  LIN {X 12449.921,Y 0.097,Z 67.094,A 90.00334,B 0.00000,C 180.00000} ; retreat
  ; Step 449, bar 1033
  LIN {X 12465.921,Y 0.097,Z 912.668,A 90.00334,B 0.00000,C 180.00000} ; outside
  LIN {X 12465.921,Y 0.097,Z 17.094,A 90.00334,B 0.00000,C 180.00000} ; preinsert
  LIN {X 12465.921,Y 0.097,Z -232.906,A 90.00334,B 0.00000,C 180.00000} ; insert
  LIN {X 12465.921,Y 0.097,Z -232.906,A 90.00334,B 0.00000,C 180.00000} ; release
  LIN {X 12465.921,Y 0.097,Z 67.094,A 90.00334,B 0.00000,C 180.00000} ; retreat
  ; Step 450, bar 295
  LIN {X 0.000,Y -2325.000,Z 1045.621,A 0.00000,B 0.00000,C 180.00000} ; outside
  LIN {X 0.000,Y -2325.000,Z 147.121,A 0.00000,B 0.00000,C 180.00000} ; preinsert
  LIN {X 0.000,Y -2325.000,Z -102.879,A 0.00000,B 0.00000,C 180.00000} ; insert
  LIN {X 0.000,Y -2325.000,Z -102.879,A 0.00000,B 0.00000,C 180.00000} ; release
  LIN {X 0.000,Y -2325.000,Z 197.121,A 0.00000,B 0.00000,C 180.00000} ; retreat
  ; Step 451, bar 322
  LIN {X 0.000,Y 2325.000,Z 1045.621,A 0.00000,B 0.00000,C 180.00000} ; outside
  LIN {X 0.000,Y 2325.000,Z 147.121,A 0.00000,B 0.00000,C 180.00000} ; preinsert
  LIN {X 0.000,Y 2325.000,Z -102.879,A 0.00000,B 0.00000,C 180.00000} ; insert
  LIN {X 0.000,Y 2325.000,Z -102.879,A 0.00000,B 0.00000,C 180.00000} ; release
  LIN {X 0.000,Y 2325.000,Z 197.121,A 0.00000,B 0.00000,C 180.00000} ; retreat
  ; Step 452, bar 293
  LIN {X 0.000,Y -1977.000,Z 1051.871,A 0.00000,B 0.00000,C 180.00000} ; outside
  LIN {X 0.000,Y -1977.000,Z 150.246,A 0.00000,B 0.00000,C 180.00000} ; preinsert
  LIN {X 0.000,Y -1977.000,Z -99.754,A 0.00000,B 0.00000,C 180.00000} ; insert
  LIN {X 0.000,Y -1977.000,Z -99.754,A 0.00000,B 0.00000,C 180.00000} ; release
  LIN {X 0.000,Y -1977.000,Z 200.246,A 0.00000,B 0.00000,C 180.00000} ; retreat
  ; Step 453, bar 320
  LIN {X 0.000,Y 1977.000,Z 1051.871,A 0.00000,B 0.00000,C 180.00000} ; outside
  LIN {X 0.000,Y 1977.000,Z 150.246,A 0.00000,B 0.00000,C 180.00000} ; preinsert
  LIN {X 0.000,Y 1977.000,Z -99.754,A 0.00000,B 0.00000,C 180.00000} ; insert
  LIN {X 0.000,Y 1977.000,Z -99.754,A 0.00000,B 0.00000,C 180.00000} ; release
  LIN {X 0.000,Y 1977.000,Z 200.246,A 0.00000,B 0.00000,C 180.00000} ; retreat
  ; Step 454, bar 294
  LIN {X 0.484,Y -2151.056,Z 1053.018,A -179.99813,B 0.00000,C 180.00000} ; outside
  LIN {X 0.484,Y -2151.056,Z 150.800,A -179.99813,B 0.00000,C 180.00000} ; preinsert
  LIN {X 0.484,Y -2151.056,Z -99.200,A -179.99813,B 0.00000,C 180.00000} ; insert
  LIN {X 0.484,Y -2151.056,Z -99.200,A -179.99813,B 0.00000,C 180.00000} ; release
  LIN {X 0.484,Y -2151.056,Z 200.800,A -179.99813,B 0.00000,C 180.00000} ; retreat
  ; Step 455, bar 1893
  LIN {X 3995.484,Y -2151.056,Z 1053.018,A -179.99813,B 0.00000,C 180.00000} ; outside
  LIN {X 3995.484,Y -2151.056,Z 150.800,A -179.99813,B 0.00000,C 180.00000} ; preinsert
  LIN {X 3995.484,Y -2151.056,Z -99.200,A -179.99813,B 0.00000,C 180.00000} ; insert
  LIN {X 3995.484,Y -2151.056,Z -99.200,A -179.99813,B 0.00000,C 180.00000} ; release
  LIN {X 3995.484,Y -2151.056,Z 200.800,A -179.99813,B 0.00000,C 180.00000} ; retreat
  ; Step 456, bar 1897
  LIN {X 7995.484,Y -2151.056,Z 1053.018,A -179.99813,B 0.00000,C 180.00000} ; outside
  LIN {X 7995.484,Y -2151.056,Z 150.800,A -179.99813,B 0.00000,C 180.00000} ; preinsert
  LIN {X 7995.484,Y -2151.056,Z -99.200,A -179.99813,B 0.00000,C 180.00000} ; insert
  LIN {X 7995.484,Y -2151.056,Z -99.200,A -179.99813,B 0.00000,C 180.00000} ; release
  LIN {X 7995.484,Y -2151.056,Z 200.800,A -179.99813,B 0.00000,C 180.00000} ; retreat
  ; Step 457, bar 1905
  LIN {X 11995.484,Y -2151.056,Z 1053.018,A -179.99813,B 0.00000,C 180.00000} ; outside
  LIN {X 11995.484,Y -2151.056,Z 150.800,A -179.99813,B 0.00000,C 180.00000} ; preinsert
  LIN {X 11995.484,Y -2151.056,Z -99.200,A -179.99813,B 0.00000,C 180.00000} ; insert
  LIN {X 11995.484,Y -2151.056,Z -99.200,A -179.99813,B 0.00000,C 180.00000} ; release
  LIN {X 11995.484,Y -2151.056,Z 200.800,A -179.99813,B 0.00000,C 180.00000} ; retreat
  ; Step 458, bar 1922
  LIN {X -11995.484,Y 2151.056,Z 1053.018,A 0.00187,B 0.00000,C 180.00000} ; outside
  LIN {X -11995.484,Y 2151.056,Z 150.800,A 0.00187,B 0.00000,C 180.00000} ; preinsert
  LIN {X -11995.484,Y 2151.056,Z -99.200,A 0.00187,B 0.00000,C 180.00000} ; insert
  LIN {X -11995.484,Y 2151.056,Z -99.200,A 0.00187,B 0.00000,C 180.00000} ; release
  LIN {X -11995.484,Y 2151.056,Z 200.800,A 0.00187,B 0.00000,C 180.00000} ; retreat
  ; Step 459, bar 1914
  LIN {X -7995.484,Y 2151.056,Z 1053.018,A 0.00187,B 0.00000,C 180.00000} ; outside
  LIN {X -7995.484,Y 2151.056,Z 150.800,A 0.00187,B 0.00000,C 180.00000} ; preinsert
  LIN {X -7995.484,Y 2151.056,Z -99.200,A 0.00187,B 0.00000,C 180.00000} ; insert
  LIN {X -7995.484,Y 2151.056,Z -99.200,A 0.00187,B 0.00000,C 180.00000} ; release
  LIN {X -7995.484,Y 2151.056,Z 200.800,A 0.00187,B 0.00000,C 180.00000} ; retreat
  ; Step 460, bar 1910
  LIN {X -3995.484,Y 2151.056,Z 1053.018,A 0.00187,B 0.00000,C 180.00000} ; outside
  LIN {X -3995.484,Y 2151.056,Z 150.800,A 0.00187,B 0.00000,C 180.00000} ; preinsert
  LIN {X -3995.484,Y 2151.056,Z -99.200,A 0.00187,B 0.00000,C 180.00000} ; insert
  LIN {X -3995.484,Y 2151.056,Z -99.200,A 0.00187,B 0.00000,C 180.00000} ; release
  LIN {X -3995.484,Y 2151.056,Z 200.800,A 0.00187,B 0.00000,C 180.00000} ; retreat
  ; Step 461, bar 1921
  LIN {X -11995.484,Y -2151.056,Z 1053.018,A -0.00187,B 0.00000,C 180.00000} ; outside
  LIN {X -11995.484,Y -2151.056,Z 150.800,A -0.00187,B 0.00000,C 180.00000} ; preinsert
  LIN {X -11995.484,Y -2151.056,Z -99.200,A -0.00187,B 0.00000,C 180.00000} ; insert
  LIN {X -11995.484,Y -2151.056,Z -99.200,A -0.00187,B 0.00000,C 180.00000} ; release
  LIN {X -11995.484,Y -2151.056,Z 200.800,A -0.00187,B 0.00000,C 180.00000} ; retreat
  ; Step 462, bar 1913
  LIN {X -7995.484,Y -2151.056,Z 1053.018,A -0.00187,B 0.00000,C 180.00000} ; outside
  LIN {X -7995.484,Y -2151.056,Z 150.800,A -0.00187,B 0.00000,C 180.00000} ; preinsert
  LIN {X -7995.484,Y -2151.056,Z -99.200,A -0.00187,B 0.00000,C 180.00000} ; insert
  LIN {X -7995.484,Y -2151.056,Z -99.200,A -0.00187,B 0.00000,C 180.00000} ; release
  LIN {X -7995.484,Y -2151.056,Z 200.800,A -0.00187,B 0.00000,C 180.00000} ; retreat
  ; Step 463, bar 1909
  LIN {X -3995.484,Y -2151.056,Z 1053.018,A -0.00187,B 0.00000,C 180.00000} ; outside
  LIN {X -3995.484,Y -2151.056,Z 150.800,A -0.00187,B 0.00000,C 180.00000} ; preinsert
  LIN {X -3995.484,Y -2151.056,Z -99.200,A -0.00187,B 0.00000,C 180.00000} ; insert
  LIN {X -3995.484,Y -2151.056,Z -99.200,A -0.00187,B 0.00000,C 180.00000} ; release
  LIN {X -3995.484,Y -2151.056,Z 200.800,A -0.00187,B 0.00000,C 180.00000} ; retreat
  ; Step 464, bar 321
  LIN {X 0.484,Y 2151.056,Z 1053.018,A 179.99813,B 0.00000,C 180.00000} ; outside
  LIN {X 0.484,Y 2151.056,Z 150.800,A 179.99813,B 0.00000,C 180.00000} ; preinsert
  LIN {X 0.484,Y 2151.056,Z -99.200,A 179.99813,B 0.00000,C 180.00000} ; insert
  LIN {X 0.484,Y 2151.056,Z -99.200,A 179.99813,B 0.00000,C 180.00000} ; release
  LIN {X 0.484,Y 2151.056,Z 200.800,A 179.99813,B 0.00000,C 180.00000} ; retreat
  ; Step 465, bar 1894
  LIN {X 3995.484,Y 2151.056,Z 1053.018,A 179.99813,B 0.00000,C 180.00000} ; outside
  LIN {X 3995.484,Y 2151.056,Z 150.800,A 179.99813,B 0.00000,C 180.00000} ; preinsert
  LIN {X 3995.484,Y 2151.056,Z -99.200,A 179.99813,B 0.00000,C 180.00000} ; insert
  LIN {X 3995.484,Y 2151.056,Z -99.200,A 179.99813,B 0.00000,C 180.00000} ; release
  LIN {X 3995.484,Y 2151.056,Z 200.800,A 179.99813,B 0.00000,C 180.00000} ; retreat
  ; Step 466, bar 1898
  LIN {X 7995.484,Y 2151.056,Z 1053.018,A 179.99813,B 0.00000,C 180.00000} ; outside
  LIN {X 7995.484,Y 2151.056,Z 150.800,A 179.99813,B 0.00000,C 180.00000} ; preinsert
  LIN {X 7995.484,Y 2151.056,Z -99.200,A 179.99813,B 0.00000,C 180.00000} ; insert
  LIN {X 7995.484,Y 2151.056,Z -99.200,A 179.99813,B 0.00000,C 180.00000} ; release
  LIN {X 7995.484,Y 2151.056,Z 200.800,A 179.99813,B 0.00000,C 180.00000} ; retreat
  ; Step 467, bar 1906
  LIN {X 11995.484,Y 2151.056,Z 1053.018,A 179.99813,B 0.00000,C 180.00000} ; outside
  LIN {X 11995.484,Y 2151.056,Z 150.800,A 179.99813,B 0.00000,C 180.00000} ; preinsert
  LIN {X 11995.484,Y 2151.056,Z -99.200,A 179.99813,B 0.00000,C 180.00000} ; insert
  LIN {X 11995.484,Y 2151.056,Z -99.200,A 179.99813,B 0.00000,C 180.00000} ; release
  LIN {X 11995.484,Y 2151.056,Z 200.800,A 179.99813,B 0.00000,C 180.00000} ; retreat
  ; Step 468, bar 1923
  LIN {X -11994.516,Y -2150.911,Z 797.364,A -179.99813,B 0.00000,C -180.00000} ; outside
  LIN {X -11994.516,Y -2150.911,Z -105.285,A -179.99813,B 0.00000,C -180.00000} ; preinsert
  LIN {X -11994.516,Y -2150.911,Z -355.285,A -179.99813,B 0.00000,C -180.00000} ; insert
  LIN {X -11994.516,Y -2150.911,Z -355.285,A -179.99813,B 0.00000,C -180.00000} ; release
  LIN {X -11994.516,Y -2150.911,Z -55.285,A -179.99813,B 0.00000,C -180.00000} ; retreat
  ; Step 469, bar 1915
  LIN {X -7994.516,Y -2150.911,Z 797.364,A -179.99813,B 0.00000,C -180.00000} ; outside
  LIN {X -7994.516,Y -2150.911,Z -105.285,A -179.99813,B 0.00000,C -180.00000} ; preinsert
  LIN {X -7994.516,Y -2150.911,Z -355.285,A -179.99813,B 0.00000,C -180.00000} ; insert
  LIN {X -7994.516,Y -2150.911,Z -355.285,A -179.99813,B 0.00000,C -180.00000} ; release
  LIN {X -7994.516,Y -2150.911,Z -55.285,A -179.99813,B 0.00000,C -180.00000} ; retreat
  ; Step 470, bar 1899
  LIN {X 7994.516,Y -2150.911,Z 797.364,A -0.00187,B 0.00000,C 180.00000} ; outside
  LIN {X 7994.516,Y -2150.911,Z -105.285,A -0.00187,B 0.00000,C 180.00000} ; preinsert
  LIN {X 7994.516,Y -2150.911,Z -355.285,A -0.00187,B 0.00000,C 180.00000} ; insert
  LIN {X 7994.516,Y -2150.911,Z -355.285,A -0.00187,B 0.00000,C 180.00000} ; release
  LIN {X 7994.516,Y -2150.911,Z -55.285,A -0.00187,B 0.00000,C 180.00000} ; retreat
  ; Step 471, bar 1907
  LIN {X 11994.516,Y -2150.911,Z 797.364,A -0.00187,B 0.00000,C 180.00000} ; outside
  LIN {X 11994.516,Y -2150.911,Z -105.285,A -0.00187,B 0.00000,C 180.00000} ; preinsert
  LIN {X 11994.516,Y -2150.911,Z -355.285,A -0.00187,B 0.00000,C 180.00000} ; insert
  LIN {X 11994.516,Y -2150.911,Z -355.285,A -0.00187,B 0.00000,C 180.00000} ; release
  LIN {X 11994.516,Y -2150.911,Z -55.285,A -0.00187,B 0.00000,C 180.00000} ; retreat
  ; Step 472, bar 1911
  LIN {X -3994.516,Y -2150.911,Z 797.364,A -179.99813,B 0.00000,C -180.00000} ; outside
  LIN {X -3994.516,Y -2150.911,Z -105.285,A -179.99813,B 0.00000,C -180.00000} ; preinsert
  LIN {X -3994.516,Y -2150.911,Z -355.285,A -179.99813,B 0.00000,C -180.00000} ; insert
  LIN {X -3994.516,Y -2150.911,Z -355.285,A -179.99813,B 0.00000,C -180.00000} ; release
  LIN {X -3994.516,Y -2150.911,Z -55.285,A -179.99813,B 0.00000,C -180.00000} ; retreat
  ; Step 473, bar 1861
  LIN {X -0.484,Y -2150.911,Z 797.364,A -0.00187,B 0.00000,C 180.00000} ; outside
  LIN {X -0.484,Y -2150.911,Z -105.285,A -0.00187,B 0.00000,C 180.00000} ; preinsert
  LIN {X -0.484,Y -2150.911,Z -355.285,A -0.00187,B 0.00000,C 180.00000} ; insert
  LIN {X -0.484,Y -2150.911,Z -355.285,A -0.00187,B 0.00000,C 180.00000} ; release
  LIN {X -0.484,Y -2150.911,Z -55.285,A -0.00187,B 0.00000,C 180.00000} ; retreat
  ; Step 474, bar 1895
  LIN {X 3994.516,Y -2150.911,Z 797.364,A -0.00187,B 0.00000,C 180.00000} ; outside
  LIN {X 3994.516,Y -2150.911,Z -105.285,A -0.00187,B 0.00000,C 180.00000} ; preinsert
  LIN {X 3994.516,Y -2150.911,Z -355.285,A -0.00187,B 0.00000,C 180.00000} ; insert
  LIN {X 3994.516,Y -2150.911,Z -355.285,A -0.00187,B 0.00000,C 180.00000} ; release
  LIN {X 3994.516,Y -2150.911,Z -55.285,A -0.00187,B 0.00000,C 180.00000} ; retreat
  ; Step 475, bar 1924
  LIN {X -11994.516,Y 2150.911,Z 797.364,A 179.99813,B 0.00000,C -180.00000} ; outside
  LIN {X -11994.516,Y 2150.911,Z -105.285,A 179.99813,B 0.00000,C -180.00000} ; preinsert
  LIN {X -11994.516,Y 2150.911,Z -355.285,A 179.99813,B 0.00000,C -180.00000} ; insert
  LIN {X -11994.516,Y 2150.911,Z -355.285,A 179.99813,B 0.00000,C -180.00000} ; release
  LIN {X -11994.516,Y 2150.911,Z -55.285,A 179.99813,B 0.00000,C -180.00000} ; retreat
  ; Step 476, bar 1916
  LIN {X -7994.516,Y 2150.911,Z 797.364,A 179.99813,B 0.00000,C -180.00000} ; outside
  LIN {X -7994.516,Y 2150.911,Z -105.285,A 179.99813,B 0.00000,C -180.00000} ; preinsert
  LIN {X -7994.516,Y 2150.911,Z -355.285,A 179.99813,B 0.00000,C -180.00000} ; insert
  LIN {X -7994.516,Y 2150.911,Z -355.285,A 179.99813,B 0.00000,C -180.00000} ; release
  LIN {X -7994.516,Y 2150.911,Z -55.285,A 179.99813,B 0.00000,C -180.00000} ; retreat
  ; Step 477, bar 1900
  LIN {X 7994.516,Y 2150.911,Z 797.364,A 0.00187,B 0.00000,C 180.00000} ; outside
  LIN {X 7994.516,Y 2150.911,Z -105.285,A 0.00187,B 0.00000,C 180.00000} ; preinsert
  LIN {X 7994.516,Y 2150.911,Z -355.285,A 0.00187,B 0.00000,C 180.00000} ; insert
  LIN {X 7994.516,Y 2150.911,Z -355.285,A 0.00187,B 0.00000,C 180.00000} ; release
  LIN {X 7994.516,Y 2150.911,Z -55.285,A 0.00187,B 0.00000,C 180.00000} ; retreat
  ; Step 478, bar 1908
  LIN {X 11994.516,Y 2150.911,Z 797.364,A 0.00187,B 0.00000,C 180.00000} ; outside
  LIN {X 11994.516,Y 2150.911,Z -105.285,A 0.00187,B 0.00000,C 180.00000} ; preinsert
  LIN {X 11994.516,Y 2150.911,Z -355.285,A 0.00187,B 0.00000,C 180.00000} ; insert
  LIN {X 11994.516,Y 2150.911,Z -355.285,A 0.00187,B 0.00000,C 180.00000} ; release
  LIN {X 11994.516,Y 2150.911,Z -55.285,A 0.00187,B 0.00000,C 180.00000} ; retreat
  ; Step 479, bar 1912
  LIN {X -3994.516,Y 2150.911,Z 797.364,A 179.99813,B 0.00000,C -180.00000} ; outside
  LIN {X -3994.516,Y 2150.911,Z -105.285,A 179.99813,B 0.00000,C -180.00000} ; preinsert
  LIN {X -3994.516,Y 2150.911,Z -355.285,A 179.99813,B 0.00000,C -180.00000} ; insert
  LIN {X -3994.516,Y 2150.911,Z -355.285,A 179.99813,B 0.00000,C -180.00000} ; release
  LIN {X -3994.516,Y 2150.911,Z -55.285,A 179.99813,B 0.00000,C -180.00000} ; retreat
  ; Step 480, bar 1874
  LIN {X -0.484,Y 2150.911,Z 797.364,A 0.00187,B 0.00000,C 180.00000} ; outside
  LIN {X -0.484,Y 2150.911,Z -105.285,A 0.00187,B 0.00000,C 180.00000} ; preinsert
  LIN {X -0.484,Y 2150.911,Z -355.285,A 0.00187,B 0.00000,C 180.00000} ; insert
  LIN {X -0.484,Y 2150.911,Z -355.285,A 0.00187,B 0.00000,C 180.00000} ; release
  LIN {X -0.484,Y 2150.911,Z -55.285,A 0.00187,B 0.00000,C 180.00000} ; retreat
  ; Step 481, bar 1896
  LIN {X 3994.516,Y 2150.911,Z 797.364,A 0.00187,B 0.00000,C 180.00000} ; outside
  LIN {X 3994.516,Y 2150.911,Z -105.285,A 0.00187,B 0.00000,C 180.00000} ; preinsert
  LIN {X 3994.516,Y 2150.911,Z -355.285,A 0.00187,B 0.00000,C 180.00000} ; insert
  LIN {X 3994.516,Y 2150.911,Z -355.285,A 0.00187,B 0.00000,C 180.00000} ; release
  LIN {X 3994.516,Y 2150.911,Z -55.285,A 0.00187,B 0.00000,C 180.00000} ; retreat
  ; Step 482, bar 1917
  LIN {X -15308.088,Y -2150.945,Z 1052.784,A -0.00257,B 0.00000,C 180.00000} ; outside
  LIN {X -15308.088,Y -2150.945,Z 150.678,A -0.00257,B 0.00000,C 180.00000} ; preinsert
  LIN {X -15308.088,Y -2150.945,Z -99.322,A -0.00257,B 0.00000,C 180.00000} ; insert
  LIN {X -15308.088,Y -2150.945,Z -99.322,A -0.00257,B 0.00000,C 180.00000} ; release
  LIN {X -15308.088,Y -2150.945,Z 200.678,A -0.00257,B 0.00000,C 180.00000} ; retreat
  ; Step 483, bar 1901
  LIN {X 15308.088,Y -2150.945,Z 1052.784,A -179.99743,B 0.00000,C 180.00000} ; outside
  LIN {X 15308.088,Y -2150.945,Z 150.678,A -179.99743,B 0.00000,C 180.00000} ; preinsert
  LIN {X 15308.088,Y -2150.945,Z -99.322,A -179.99743,B 0.00000,C 180.00000} ; insert
  LIN {X 15308.088,Y -2150.945,Z -99.322,A -179.99743,B 0.00000,C 180.00000} ; release
  LIN {X 15308.088,Y -2150.945,Z 200.678,A -179.99743,B 0.00000,C 180.00000} ; retreat
  ; Step 484, bar 1918
  LIN {X -15308.088,Y 2150.945,Z 1052.784,A 0.00257,B 0.00000,C 180.00000} ; outside
  LIN {X -15308.088,Y 2150.945,Z 150.678,A 0.00257,B 0.00000,C 180.00000} ; preinsert
  LIN {X -15308.088,Y 2150.945,Z -99.322,A 0.00257,B 0.00000,C 180.00000} ; insert
  LIN {X -15308.088,Y 2150.945,Z -99.322,A 0.00257,B 0.00000,C 180.00000} ; release
  LIN {X -15308.088,Y 2150.945,Z 200.678,A 0.00257,B 0.00000,C 180.00000} ; retreat
  ; Step 485, bar 1902
  LIN {X 15308.088,Y 2150.945,Z 1052.784,A 179.99743,B 0.00000,C -180.00000} ; outside
  LIN {X 15308.088,Y 2150.945,Z 150.678,A 179.99743,B 0.00000,C -180.00000} ; preinsert
  LIN {X 15308.088,Y 2150.945,Z -99.322,A 179.99743,B 0.00000,C -180.00000} ; insert
  LIN {X 15308.088,Y 2150.945,Z -99.322,A 179.99743,B 0.00000,C -180.00000} ; release
  LIN {X 15308.088,Y 2150.945,Z 200.678,A 179.99743,B 0.00000,C -180.00000} ; retreat
  ; Step 486, bar 1852
  LIN {X -16250.000,Y -0.156,Z 909.110,A 90.00000,B 0.00000,C 180.00000} ; outside
  LIN {X -16250.000,Y -0.156,Z 7.730,A 90.00000,B 0.00000,C 180.00000} ; preinsert
  LIN {X -16250.000,Y -0.156,Z -242.270,A 90.00000,B 0.00000,C 180.00000} ; insert
  LIN {X -16250.000,Y -0.156,Z -242.270,A 90.00000,B 0.00000,C 180.00000} ; release
  LIN {X -16250.000,Y -0.156,Z 57.730,A 90.00000,B 0.00000,C 180.00000} ; retreat
  ; Step 487, bar 1851
  LIN {X -16150.000,Y -0.156,Z 909.110,A 90.00000,B 0.00000,C 180.00000} ; outside
  LIN {X -16150.000,Y -0.156,Z 7.730,A 90.00000,B 0.00000,C 180.00000} ; preinsert
  LIN {X -16150.000,Y -0.156,Z -242.270,A 90.00000,B 0.00000,C 180.00000} ; insert
  LIN {X -16150.000,Y -0.156,Z -242.270,A 90.00000,B 0.00000,C 180.00000} ; release
  LIN {X -16150.000,Y -0.156,Z 57.730,A 90.00000,B 0.00000,C 180.00000} ; retreat
  ; Step 488, bar 1064
  LIN {X 16150.000,Y -0.171,Z 909.110,A 90.00000,B 0.00000,C 180.00000} ; outside
  LIN {X 16150.000,Y -0.171,Z 7.730,A 90.00000,B 0.00000,C 180.00000} ; preinsert
  LIN {X 16150.000,Y -0.171,Z -242.270,A 90.00000,B 0.00000,C 180.00000} ; insert
  LIN {X 16150.000,Y -0.171,Z -242.270,A 90.00000,B 0.00000,C 180.00000} ; release
  LIN {X 16150.000,Y -0.171,Z 57.730,A 90.00000,B 0.00000,C 180.00000} ; retreat
  ; Step 489, bar 1065
  LIN {X 16250.000,Y -0.171,Z 909.110,A 90.00000,B 0.00000,C 180.00000} ; outside
  LIN {X 16250.000,Y -0.171,Z 7.730,A 90.00000,B 0.00000,C 180.00000} ; preinsert
  LIN {X 16250.000,Y -0.171,Z -242.270,A 90.00000,B 0.00000,C 180.00000} ; insert
  LIN {X 16250.000,Y -0.171,Z -242.270,A 90.00000,B 0.00000,C 180.00000} ; release
  LIN {X 16250.000,Y -0.171,Z 57.730,A 90.00000,B 0.00000,C 180.00000} ; retreat
  ; Step 490, bar 1233
  LIN {X -12349.921,Y 0.110,Z 926.030,A 89.99666,B 0.00000,C 180.00000} ; outside
  LIN {X -12349.921,Y 0.110,Z 23.775,A 89.99666,B 0.00000,C 180.00000} ; preinsert
  LIN {X -12349.921,Y 0.110,Z -226.225,A 89.99666,B 0.00000,C 180.00000} ; insert
  LIN {X -12349.921,Y 0.110,Z -226.225,A 89.99666,B 0.00000,C 180.00000} ; release
  LIN {X -12349.921,Y 0.110,Z 73.775,A 89.99666,B 0.00000,C 180.00000} ; retreat
  ; Step 491, bar 1018
  LIN {X 12349.921,Y 0.097,Z 926.030,A 90.00334,B 0.00000,C 180.00000} ; outside
  LIN {X 12349.921,Y 0.097,Z 23.775,A 90.00334,B 0.00000,C 180.00000} ; preinsert
  LIN {X 12349.921,Y 0.097,Z -226.225,A 90.00334,B 0.00000,C 180.00000} ; insert
  LIN {X 12349.921,Y 0.097,Z -226.225,A 90.00334,B 0.00000,C 180.00000} ; release
  LIN {X 12349.921,Y 0.097,Z 73.775,A 90.00334,B 0.00000,C 180.00000} ; retreat
  ; Step 492, bar 2977
  LIN {X -14850.007,Y -1181.237,Z 942.517,A -92.05282,B 0.00000,C -180.00000} ; outside
  LIN {X -14850.007,Y -1181.237,Z 3.500,A -92.05282,B 0.00000,C -180.00000} ; preinsert
  LIN {X -14850.007,Y -1181.237,Z -246.500,A -92.05282,B 0.00000,C -180.00000} ; insert
  LIN {X -14850.007,Y -1181.237,Z -246.500,A -92.05282,B 0.00000,C -180.00000} ; release
  LIN {X -14850.007,Y -1181.237,Z 53.500,A -92.05282,B 0.00000,C -180.00000} ; retreat
  ; Step 493, bar 3016
  LIN {X 14850.007,Y -1181.237,Z 942.518,A -87.94718,B 0.00000,C 180.00000} ; outside
  LIN {X 14850.007,Y -1181.237,Z 3.500,A -87.94718,B 0.00000,C 180.00000} ; preinsert
  LIN {X 14850.007,Y -1181.237,Z -246.500,A -87.94718,B 0.00000,C 180.00000} ; insert
  LIN {X 14850.007,Y -1181.237,Z -246.500,A -87.94718,B 0.00000,C 180.00000} ; release
  LIN {X 14850.007,Y -1181.237,Z 53.500,A -87.94718,B 0.00000,C 180.00000} ; retreat
  ; Step 494, bar 2959
  LIN {X -14850.007,Y 1181.237,Z 942.518,A 92.05282,B 0.00000,C 180.00000} ; outside
  LIN {X -14850.007,Y 1181.237,Z 3.500,A 92.05282,B 0.00000,C 180.00000} ; preinsert
  LIN {X -14850.007,Y 1181.237,Z -246.500,A 92.05282,B 0.00000,C 180.00000} ; insert
  LIN {X -14850.007,Y 1181.237,Z -246.500,A 92.05282,B 0.00000,C 180.00000} ; release
  LIN {X -14850.007,Y 1181.237,Z 53.500,A 92.05282,B 0.00000,C 180.00000} ; retreat
  ; Step 495, bar 2998
  LIN {X 14850.007,Y 1181.237,Z 942.517,A 87.94718,B 0.00000,C 180.00000} ; outside
  LIN {X 14850.007,Y 1181.237,Z 3.500,A 87.94718,B 0.00000,C 180.00000} ; preinsert
  LIN {X 14850.007,Y 1181.237,Z -246.500,A 87.94718,B 0.00000,C 180.00000} ; insert
  LIN {X 14850.007,Y 1181.237,Z -246.500,A 87.94718,B 0.00000,C 180.00000} ; release
  LIN {X 14850.007,Y 1181.237,Z 53.500,A 87.94718,B 0.00000,C 180.00000} ; retreat
  ; Step 496, bar 3011
  LIN {X 14050.059,Y -1181.145,Z 931.267,A 88.24449,B 0.00000,C 180.00000} ; outside
  LIN {X 14050.059,Y -1181.145,Z 14.532,A 88.24449,B 0.00000,C 180.00000} ; preinsert
  LIN {X 14050.059,Y -1181.145,Z -235.468,A 88.24449,B 0.00000,C 180.00000} ; insert
  LIN {X 14050.059,Y -1181.145,Z -235.468,A 88.24449,B 0.00000,C 180.00000} ; release
  LIN {X 14050.059,Y -1181.145,Z 64.532,A 88.24449,B 0.00000,C 180.00000} ; retreat
  ; Step 497, bar 2953
  LIN {X -14050.059,Y 1181.145,Z 931.267,A -91.75551,B 0.00000,C -180.00000} ; outside
  LIN {X -14050.059,Y 1181.145,Z 14.532,A -91.75551,B 0.00000,C -180.00000} ; preinsert
  LIN {X -14050.059,Y 1181.145,Z -235.468,A -91.75551,B 0.00000,C -180.00000} ; insert
  LIN {X -14050.059,Y 1181.145,Z -235.468,A -91.75551,B 0.00000,C -180.00000} ; release
  LIN {X -14050.059,Y 1181.145,Z 64.532,A -91.75551,B 0.00000,C -180.00000} ; retreat
  ; Step 498, bar 2972
  LIN {X -14050.059,Y -1181.145,Z 931.267,A 91.75551,B 0.00000,C 180.00000} ; outside
  LIN {X -14050.059,Y -1181.145,Z 14.532,A 91.75551,B 0.00000,C 180.00000} ; preinsert
  LIN {X -14050.059,Y -1181.145,Z -235.468,A 91.75551,B 0.00000,C 180.00000} ; insert
  LIN {X -14050.059,Y -1181.145,Z -235.468,A 91.75551,B 0.00000,C 180.00000} ; release
  LIN {X -14050.059,Y -1181.145,Z 64.532,A 91.75551,B 0.00000,C 180.00000} ; retreat
  ; Step 499, bar 2992
  LIN {X 14050.059,Y 1181.145,Z 931.267,A -88.24449,B 0.00000,C 180.00000} ; outside
  LIN {X 14050.059,Y 1181.145,Z 14.532,A -88.24449,B 0.00000,C 180.00000} ; preinsert
  LIN {X 14050.059,Y 1181.145,Z -235.468,A -88.24449,B 0.00000,C 180.00000} ; insert
  LIN {X 14050.059,Y 1181.145,Z -235.468,A -88.24449,B 0.00000,C 180.00000} ; release
  LIN {X 14050.059,Y 1181.145,Z 64.532,A -88.24449,B 0.00000,C 180.00000} ; retreat
  ; Step 500, bar 2967
  LIN {X -13249.916,Y -1181.296,Z 955.534,A 87.44234,B 0.00000,C -180.00000} ; outside
  LIN {X -13249.916,Y -1181.296,Z 50.876,A 87.44234,B 0.00000,C -180.00000} ; preinsert
  LIN {X -13249.916,Y -1181.296,Z -199.124,A 87.44234,B 0.00000,C -180.00000} ; insert
  LIN {X -13249.916,Y -1181.296,Z -199.124,A 87.44234,B 0.00000,C -180.00000} ; release
  LIN {X -13249.916,Y -1181.296,Z 100.876,A 87.44234,B 0.00000,C -180.00000} ; retreat
  ; Step 501, bar 2986
  LIN {X 13249.916,Y 1181.296,Z 955.534,A -92.55766,B 0.00000,C -180.00000} ; outside
  LIN {X 13249.916,Y 1181.296,Z 50.876,A -92.55766,B 0.00000,C -180.00000} ; preinsert
  LIN {X 13249.916,Y 1181.296,Z -199.124,A -92.55766,B 0.00000,C -180.00000} ; insert
  LIN {X 13249.916,Y 1181.296,Z -199.124,A -92.55766,B 0.00000,C -180.00000} ; release
  LIN {X 13249.916,Y 1181.296,Z 100.876,A -92.55766,B 0.00000,C -180.00000} ; retreat
  ; Step 502, bar 3006
  LIN {X 13249.916,Y -1181.296,Z 955.534,A 92.55766,B 0.00000,C 180.00000} ; outside
  LIN {X 13249.916,Y -1181.296,Z 50.876,A 92.55766,B 0.00000,C 180.00000} ; preinsert
  LIN {X 13249.916,Y -1181.296,Z -199.124,A 92.55766,B 0.00000,C 180.00000} ; insert
  LIN {X 13249.916,Y -1181.296,Z -199.124,A 92.55766,B 0.00000,C 180.00000} ; release
  LIN {X 13249.916,Y -1181.296,Z 100.876,A 92.55766,B 0.00000,C 180.00000} ; retreat
  ; Step 503, bar 2947
  LIN {X -13249.916,Y 1181.296,Z 955.534,A -87.44234,B 0.00000,C -180.00000} ; outside
  LIN {X -13249.916,Y 1181.296,Z 50.876,A -87.44234,B 0.00000,C -180.00000} ; preinsert
  LIN {X -13249.916,Y 1181.296,Z -199.124,A -87.44234,B 0.00000,C -180.00000} ; insert
  LIN {X -13249.916,Y 1181.296,Z -199.124,A -87.44234,B 0.00000,C -180.00000} ; release
  LIN {X -13249.916,Y 1181.296,Z 100.876,A -87.44234,B 0.00000,C -180.00000} ; retreat
  ; Step 504, bar 292
  LIN {X 0.000,Y -1823.000,Z 1065.621,A 0.00000,B 0.00000,C 180.00000} ; outside
  LIN {X 0.000,Y -1823.000,Z 157.121,A 0.00000,B 0.00000,C 180.00000} ; preinsert
  LIN {X 0.000,Y -1823.000,Z -92.879,A 0.00000,B 0.00000,C 180.00000} ; insert
  LIN {X 0.000,Y -1823.000,Z -92.879,A 0.00000,B 0.00000,C 180.00000} ; release
  LIN {X 0.000,Y -1823.000,Z 207.121,A 0.00000,B 0.00000,C 180.00000} ; retreat
  ; Step 505, bar 319
  LIN {X 0.000,Y 1823.000,Z 1065.621,A 0.00000,B 0.00000,C 180.00000} ; outside
  LIN {X 0.000,Y 1823.000,Z 157.121,A 0.00000,B 0.00000,C 180.00000} ; preinsert
  LIN {X 0.000,Y 1823.000,Z -92.879,A 0.00000,B 0.00000,C 180.00000} ; insert
  LIN {X 0.000,Y 1823.000,Z -92.879,A 0.00000,B 0.00000,C 180.00000} ; release
  LIN {X 0.000,Y 1823.000,Z 207.121,A 0.00000,B 0.00000,C 180.00000} ; retreat
  ; Step 506, bar 291
  LIN {X 0.000,Y -1669.000,Z 1071.871,A 0.00000,B 0.00000,C 180.00000} ; outside
  LIN {X 0.000,Y -1669.000,Z 160.246,A 0.00000,B 0.00000,C 180.00000} ; preinsert
  LIN {X 0.000,Y -1669.000,Z -89.754,A 0.00000,B 0.00000,C 180.00000} ; insert
  LIN {X 0.000,Y -1669.000,Z -89.754,A 0.00000,B 0.00000,C 180.00000} ; release
  LIN {X 0.000,Y -1669.000,Z 210.246,A 0.00000,B 0.00000,C 180.00000} ; retreat
  ; Step 507, bar 318
  LIN {X 0.000,Y 1669.000,Z 1071.871,A 0.00000,B 0.00000,C 180.00000} ; outside
  LIN {X 0.000,Y 1669.000,Z 160.246,A 0.00000,B 0.00000,C 180.00000} ; preinsert
  LIN {X 0.000,Y 1669.000,Z -89.754,A 0.00000,B 0.00000,C 180.00000} ; insert
  LIN {X 0.000,Y 1669.000,Z -89.754,A 0.00000,B 0.00000,C 180.00000} ; release
  LIN {X 0.000,Y 1669.000,Z 210.246,A 0.00000,B 0.00000,C 180.00000} ; retreat
  ; Step 508, bar 1232
  LIN {X -12249.921,Y 0.110,Z 947.280,A 89.99666,B 0.00000,C 180.00000} ; outside
  LIN {X -12249.921,Y 0.110,Z 34.400,A 89.99666,B 0.00000,C 180.00000} ; preinsert
  LIN {X -12249.921,Y 0.110,Z -215.600,A 89.99666,B 0.00000,C 180.00000} ; insert
  LIN {X -12249.921,Y 0.110,Z -215.600,A 89.99666,B 0.00000,C 180.00000} ; release
  LIN {X -12249.921,Y 0.110,Z 84.400,A 89.99666,B 0.00000,C 180.00000} ; retreat
  ; Step 509, bar 1229
  LIN {X -12124.921,Y 0.110,Z 947.280,A 89.99666,B 0.00000,C 180.00000} ; outside
  LIN {X -12124.921,Y 0.110,Z 34.400,A 89.99666,B 0.00000,C 180.00000} ; preinsert
  LIN {X -12124.921,Y 0.110,Z -215.600,A 89.99666,B 0.00000,C 180.00000} ; insert
  LIN {X -12124.921,Y 0.110,Z -215.600,A 89.99666,B 0.00000,C 180.00000} ; release
  LIN {X -12124.921,Y 0.110,Z 84.400,A 89.99666,B 0.00000,C 180.00000} ; retreat
  ; Step 510, bar 1231
  LIN {X -12015.921,Y 0.110,Z 947.280,A 89.99666,B 0.00000,C 180.00000} ; outside
  LIN {X -12015.921,Y 0.110,Z 34.400,A 89.99666,B 0.00000,C 180.00000} ; preinsert
  LIN {X -12015.921,Y 0.110,Z -215.600,A 89.99666,B 0.00000,C 180.00000} ; insert
  LIN {X -12015.921,Y 0.110,Z -215.600,A 89.99666,B 0.00000,C 180.00000} ; release
  LIN {X -12015.921,Y 0.110,Z 84.400,A 89.99666,B 0.00000,C 180.00000} ; retreat
  ; Step 511, bar 1230
  LIN {X -11999.921,Y 0.110,Z 947.280,A 89.99666,B 0.00000,C 180.00000} ; outside
  LIN {X -11999.921,Y 0.110,Z 34.400,A 89.99666,B 0.00000,C 180.00000} ; preinsert
  LIN {X -11999.921,Y 0.110,Z -215.600,A 89.99666,B 0.00000,C 180.00000} ; insert
  LIN {X -11999.921,Y 0.110,Z -215.600,A 89.99666,B 0.00000,C 180.00000} ; release
  LIN {X -11999.921,Y 0.110,Z 84.400,A 89.99666,B 0.00000,C 180.00000} ; retreat
  ; Step 512, bar 1228
  LIN {X -11874.921,Y 0.110,Z 947.280,A 89.99666,B 0.00000,C 180.00000} ; outside
  LIN {X -11874.921,Y 0.110,Z 34.400,A 89.99666,B 0.00000,C 180.00000} ; preinsert
  LIN {X -11874.921,Y 0.110,Z -215.600,A 89.99666,B 0.00000,C 180.00000} ; insert
  LIN {X -11874.921,Y 0.110,Z -215.600,A 89.99666,B 0.00000,C 180.00000} ; release
  LIN {X -11874.921,Y 0.110,Z 84.400,A 89.99666,B 0.00000,C 180.00000} ; retreat
  ; Step 513, bar 1227
  LIN {X -11749.921,Y 0.110,Z 947.280,A 89.99666,B 0.00000,C 180.00000} ; outside
  LIN {X -11749.921,Y 0.110,Z 34.400,A 89.99666,B 0.00000,C 180.00000} ; preinsert
  LIN {X -11749.921,Y 0.110,Z -215.600,A 89.99666,B 0.00000,C 180.00000} ; insert
  LIN {X -11749.921,Y 0.110,Z -215.600,A 89.99666,B 0.00000,C 180.00000} ; release
  LIN {X -11749.921,Y 0.110,Z 84.400,A 89.99666,B 0.00000,C 180.00000} ; retreat
  ; Step 514, bar 1224
  LIN {X -11624.921,Y 0.110,Z 947.280,A 89.99666,B 0.00000,C 180.00000} ; outside
  LIN {X -11624.921,Y 0.110,Z 34.400,A 89.99666,B 0.00000,C 180.00000} ; preinsert
  LIN {X -11624.921,Y 0.110,Z -215.600,A 89.99666,B 0.00000,C 180.00000} ; insert
  LIN {X -11624.921,Y 0.110,Z -215.600,A 89.99666,B 0.00000,C 180.00000} ; release
  LIN {X -11624.921,Y 0.110,Z 84.400,A 89.99666,B 0.00000,C 180.00000} ; retreat
  ; Step 515, bar 1226
  LIN {X -11515.921,Y 0.110,Z 947.280,A 89.99666,B 0.00000,C 180.00000} ; outside
  LIN {X -11515.921,Y 0.110,Z 34.400,A 89.99666,B 0.00000,C 180.00000} ; preinsert
  LIN {X -11515.921,Y 0.110,Z -215.600,A 89.99666,B 0.00000,C 180.00000} ; insert
  LIN {X -11515.921,Y 0.110,Z -215.600,A 89.99666,B 0.00000,C 180.00000} ; release
  LIN {X -11515.921,Y 0.110,Z 84.400,A 89.99666,B 0.00000,C 180.00000} ; retreat
  ; Step 516, bar 1225
  LIN {X -11499.921,Y 0.110,Z 947.280,A 89.99666,B 0.00000,C 180.00000} ; outside
  LIN {X -11499.921,Y 0.110,Z 34.400,A 89.99666,B 0.00000,C 180.00000} ; preinsert
  LIN {X -11499.921,Y 0.110,Z -215.600,A 89.99666,B 0.00000,C 180.00000} ; insert
  LIN {X -11499.921,Y 0.110,Z -215.600,A 89.99666,B 0.00000,C 180.00000} ; release
  LIN {X -11499.921,Y 0.110,Z 84.400,A 89.99666,B 0.00000,C 180.00000} ; retreat
  ; Step 517, bar 1223
  LIN {X -11374.921,Y 0.110,Z 947.280,A 89.99666,B 0.00000,C 180.00000} ; outside
  LIN {X -11374.921,Y 0.110,Z 34.400,A 89.99666,B 0.00000,C 180.00000} ; preinsert
  LIN {X -11374.921,Y 0.110,Z -215.600,A 89.99666,B 0.00000,C 180.00000} ; insert
  LIN {X -11374.921,Y 0.110,Z -215.600,A 89.99666,B 0.00000,C 180.00000} ; release
  LIN {X -11374.921,Y 0.110,Z 84.400,A 89.99666,B 0.00000,C 180.00000} ; retreat
  ; Step 518, bar 1222
  LIN {X -11249.921,Y 0.110,Z 947.280,A 89.99666,B 0.00000,C 180.00000} ; outside
  LIN {X -11249.921,Y 0.110,Z 34.400,A 89.99666,B 0.00000,C 180.00000} ; preinsert
  LIN {X -11249.921,Y 0.110,Z -215.600,A 89.99666,B 0.00000,C 180.00000} ; insert
  LIN {X -11249.921,Y 0.110,Z -215.600,A 89.99666,B 0.00000,C 180.00000} ; release
  LIN {X -11249.921,Y 0.110,Z 84.400,A 89.99666,B 0.00000,C 180.00000} ; retreat
  ; Step 519, bar 1219
  LIN {X -11124.921,Y 0.110,Z 947.280,A 89.99666,B 0.00000,C 180.00000} ; outside
  LIN {X -11124.921,Y 0.110,Z 34.400,A 89.99666,B 0.00000,C 180.00000} ; preinsert
  LIN {X -11124.921,Y 0.110,Z -215.600,A 89.99666,B 0.00000,C 180.00000} ; insert
  LIN {X -11124.921,Y 0.110,Z -215.600,A 89.99666,B 0.00000,C 180.00000} ; release
  LIN {X -11124.921,Y 0.110,Z 84.400,A 89.99666,B 0.00000,C 180.00000} ; retreat
  ; Step 520, bar 1221
  LIN {X -11015.921,Y 0.110,Z 947.280,A 89.99666,B 0.00000,C 180.00000} ; outside
  LIN {X -11015.921,Y 0.110,Z 34.400,A 89.99666,B 0.00000,C 180.00000} ; preinsert
  LIN {X -11015.921,Y 0.110,Z -215.600,A 89.99666,B 0.00000,C 180.00000} ; insert
  LIN {X -11015.921,Y 0.110,Z -215.600,A 89.99666,B 0.00000,C 180.00000} ; release
  LIN {X -11015.921,Y 0.110,Z 84.400,A 89.99666,B 0.00000,C 180.00000} ; retreat
  ; Step 521, bar 1220
  LIN {X -10999.921,Y 0.110,Z 947.280,A 89.99666,B 0.00000,C 180.00000} ; outside
  LIN {X -10999.921,Y 0.110,Z 34.400,A 89.99666,B 0.00000,C 180.00000} ; preinsert
  LIN {X -10999.921,Y 0.110,Z -215.600,A 89.99666,B 0.00000,C 180.00000} ; insert
  LIN {X -10999.921,Y 0.110,Z -215.600,A 89.99666,B 0.00000,C 180.00000} ; release
  LIN {X -10999.921,Y 0.110,Z 84.400,A 89.99666,B 0.00000,C 180.00000} ; retreat
  ; Step 522, bar 1218
  LIN {X -10874.921,Y 0.110,Z 947.280,A 89.99666,B 0.00000,C 180.00000} ; outside
  LIN {X -10874.921,Y 0.110,Z 34.400,A 89.99666,B 0.00000,C 180.00000} ; preinsert
  LIN {X -10874.921,Y 0.110,Z -215.600,A 89.99666,B 0.00000,C 180.00000} ; insert
  LIN {X -10874.921,Y 0.110,Z -215.600,A 89.99666,B 0.00000,C 180.00000} ; release
  LIN {X -10874.921,Y 0.110,Z 84.400,A 89.99666,B 0.00000,C 180.00000} ; retreat
  ; Step 523, bar 1217
  LIN {X -10749.921,Y 0.110,Z 947.280,A 89.99666,B 0.00000,C 180.00000} ; outside
  LIN {X -10749.921,Y 0.110,Z 34.400,A 89.99666,B 0.00000,C 180.00000} ; preinsert
  LIN {X -10749.921,Y 0.110,Z -215.600,A 89.99666,B 0.00000,C 180.00000} ; insert
  LIN {X -10749.921,Y 0.110,Z -215.600,A 89.99666,B 0.00000,C 180.00000} ; release
  LIN {X -10749.921,Y 0.110,Z 84.400,A 89.99666,B 0.00000,C 180.00000} ; retreat
  ; Step 524, bar 1214
  LIN {X -10624.921,Y 0.110,Z 947.280,A 89.99666,B 0.00000,C 180.00000} ; outside
  LIN {X -10624.921,Y 0.110,Z 34.400,A 89.99666,B 0.00000,C 180.00000} ; preinsert
  LIN {X -10624.921,Y 0.110,Z -215.600,A 89.99666,B 0.00000,C 180.00000} ; insert
  LIN {X -10624.921,Y 0.110,Z -215.600,A 89.99666,B 0.00000,C 180.00000} ; release
  LIN {X -10624.921,Y 0.110,Z 84.400,A 89.99666,B 0.00000,C 180.00000} ; retreat
  ; Step 525, bar 1216
  LIN {X -10515.921,Y 0.110,Z 947.280,A 89.99666,B 0.00000,C 180.00000} ; outside
  LIN {X -10515.921,Y 0.110,Z 34.400,A 89.99666,B 0.00000,C 180.00000} ; preinsert
  LIN {X -10515.921,Y 0.110,Z -215.600,A 89.99666,B 0.00000,C 180.00000} ; insert
  LIN {X -10515.921,Y 0.110,Z -215.600,A 89.99666,B 0.00000,C 180.00000} ; release
  LIN {X -10515.921,Y 0.110,Z 84.400,A 89.99666,B 0.00000,C 180.00000} ; retreat
  ; Step 526, bar 1215
  LIN {X -10499.921,Y 0.110,Z 947.280,A 89.99666,B 0.00000,C 180.00000} ; outside
  LIN {X -10499.921,Y 0.110,Z 34.400,A 89.99666,B 0.00000,C 180.00000} ; preinsert
  LIN {X -10499.921,Y 0.110,Z -215.600,A 89.99666,B 0.00000,C 180.00000} ; insert
  LIN {X -10499.921,Y 0.110,Z -215.600,A 89.99666,B 0.00000,C 180.00000} ; release
  LIN {X -10499.921,Y 0.110,Z 84.400,A 89.99666,B 0.00000,C 180.00000} ; retreat
  ; Step 527, bar 1213
  LIN {X -10374.921,Y 0.110,Z 947.280,A 89.99666,B 0.00000,C 180.00000} ; outside
  LIN {X -10374.921,Y 0.110,Z 34.400,A 89.99666,B 0.00000,C 180.00000} ; preinsert
  LIN {X -10374.921,Y 0.110,Z -215.600,A 89.99666,B 0.00000,C 180.00000} ; insert
  LIN {X -10374.921,Y 0.110,Z -215.600,A 89.99666,B 0.00000,C 180.00000} ; release
  LIN {X -10374.921,Y 0.110,Z 84.400,A 89.99666,B 0.00000,C 180.00000} ; retreat
  ; Step 528, bar 1212
  LIN {X -10249.921,Y 0.110,Z 947.280,A 89.99666,B 0.00000,C 180.00000} ; outside
  LIN {X -10249.921,Y 0.110,Z 34.400,A 89.99666,B 0.00000,C 180.00000} ; preinsert
  LIN {X -10249.921,Y 0.110,Z -215.600,A 89.99666,B 0.00000,C 180.00000} ; insert
  LIN {X -10249.921,Y 0.110,Z -215.600,A 89.99666,B 0.00000,C 180.00000} ; release
  LIN {X -10249.921,Y 0.110,Z 84.400,A 89.99666,B 0.00000,C 180.00000} ; retreat
  ; Step 529, bar 1209
  LIN {X -10124.921,Y 0.110,Z 947.280,A 89.99666,B 0.00000,C 180.00000} ; outside
  LIN {X -10124.921,Y 0.110,Z 34.400,A 89.99666,B 0.00000,C 180.00000} ; preinsert
  LIN {X -10124.921,Y 0.110,Z -215.600,A 89.99666,B 0.00000,C 180.00000} ; insert
  LIN {X -10124.921,Y 0.110,Z -215.600,A 89.99666,B 0.00000,C 180.00000} ; release
  LIN {X -10124.921,Y 0.110,Z 84.400,A 89.99666,B 0.00000,C 180.00000} ; retreat
  ; Step 530, bar 1208
  LIN {X -9999.921,Y 0.110,Z 947.280,A 89.99666,B 0.00000,C 180.00000} ; outside
  LIN {X -9999.921,Y 0.110,Z 34.400,A 89.99666,B 0.00000,C 180.00000} ; preinsert
  LIN {X -9999.921,Y 0.110,Z -215.600,A 89.99666,B 0.00000,C 180.00000} ; insert
  LIN {X -9999.921,Y 0.110,Z -215.600,A 89.99666,B 0.00000,C 180.00000} ; release
  LIN {X -9999.921,Y 0.110,Z 84.400,A 89.99666,B 0.00000,C 180.00000} ; retreat
  ; Step 531, bar 1211
  LIN {X -9890.921,Y 0.110,Z 947.280,A 89.99666,B 0.00000,C 180.00000} ; outside
  LIN {X -9890.921,Y 0.110,Z 34.400,A 89.99666,B 0.00000,C 180.00000} ; preinsert
  LIN {X -9890.921,Y 0.110,Z -215.600,A 89.99666,B 0.00000,C 180.00000} ; insert
  LIN {X -9890.921,Y 0.110,Z -215.600,A 89.99666,B 0.00000,C 180.00000} ; release
  LIN {X -9890.921,Y 0.110,Z 84.400,A 89.99666,B 0.00000,C 180.00000} ; retreat
  ; Step 532, bar 1210
  LIN {X -9874.921,Y 0.110,Z 947.280,A 89.99666,B 0.00000,C 180.00000} ; outside
  LIN {X -9874.921,Y 0.110,Z 34.400,A 89.99666,B 0.00000,C 180.00000} ; preinsert
  LIN {X -9874.921,Y 0.110,Z -215.600,A 89.99666,B 0.00000,C 180.00000} ; insert
  LIN {X -9874.921,Y 0.110,Z -215.600,A 89.99666,B 0.00000,C 180.00000} ; release
  LIN {X -9874.921,Y 0.110,Z 84.400,A 89.99666,B 0.00000,C 180.00000} ; retreat
  ; Step 533, bar 1207
  LIN {X -9749.921,Y 0.110,Z 947.280,A 89.99666,B 0.00000,C 180.00000} ; outside
  LIN {X -9749.921,Y 0.110,Z 34.400,A 89.99666,B 0.00000,C 180.00000} ; preinsert
  LIN {X -9749.921,Y 0.110,Z -215.600,A 89.99666,B 0.00000,C 180.00000} ; insert
  LIN {X -9749.921,Y 0.110,Z -215.600,A 89.99666,B 0.00000,C 180.00000} ; release
  LIN {X -9749.921,Y 0.110,Z 84.400,A 89.99666,B 0.00000,C 180.00000} ; retreat
  ; Step 534, bar 1204
  LIN {X -9624.921,Y 0.110,Z 947.280,A 89.99666,B 0.00000,C 180.00000} ; outside
  LIN {X -9624.921,Y 0.110,Z 34.400,A 89.99666,B 0.00000,C 180.00000} ; preinsert
  LIN {X -9624.921,Y 0.110,Z -215.600,A 89.99666,B 0.00000,C 180.00000} ; insert
  LIN {X -9624.921,Y 0.110,Z -215.600,A 89.99666,B 0.00000,C 180.00000} ; release
  LIN {X -9624.921,Y 0.110,Z 84.400,A 89.99666,B 0.00000,C 180.00000} ; retreat
  ; Step 535, bar 1206
  LIN {X -9515.921,Y 0.110,Z 947.280,A 89.99666,B 0.00000,C 180.00000} ; outside
  LIN {X -9515.921,Y 0.110,Z 34.400,A 89.99666,B 0.00000,C 180.00000} ; preinsert
  LIN {X -9515.921,Y 0.110,Z -215.600,A 89.99666,B 0.00000,C 180.00000} ; insert
  LIN {X -9515.921,Y 0.110,Z -215.600,A 89.99666,B 0.00000,C 180.00000} ; release
  LIN {X -9515.921,Y 0.110,Z 84.400,A 89.99666,B 0.00000,C 180.00000} ; retreat
  ; Step 536, bar 1205
  LIN {X -9499.921,Y 0.110,Z 947.280,A 89.99666,B 0.00000,C 180.00000} ; outside
  LIN {X -9499.921,Y 0.110,Z 34.400,A 89.99666,B 0.00000,C 180.00000} ; preinsert
  LIN {X -9499.921,Y 0.110,Z -215.600,A 89.99666,B 0.00000,C 180.00000} ; insert
  LIN {X -9499.921,Y 0.110,Z -215.600,A 89.99666,B 0.00000,C 180.00000} ; release
  LIN {X -9499.921,Y 0.110,Z 84.400,A 89.99666,B 0.00000,C 180.00000} ; retreat
  ; Step 537, bar 1203
  LIN {X -9374.921,Y 0.110,Z 947.280,A 89.99666,B 0.00000,C 180.00000} ; outside
  LIN {X -9374.921,Y 0.110,Z 34.400,A 89.99666,B 0.00000,C 180.00000} ; preinsert
  LIN {X -9374.921,Y 0.110,Z -215.600,A 89.99666,B 0.00000,C 180.00000} ; insert
  LIN {X -9374.921,Y 0.110,Z -215.600,A 89.99666,B 0.00000,C 180.00000} ; release
  LIN {X -9374.921,Y 0.110,Z 84.400,A 89.99666,B 0.00000,C 180.00000} ; retreat
  ; Step 538, bar 1202
  LIN {X -9249.921,Y 0.110,Z 947.280,A 89.99666,B 0.00000,C 180.00000} ; outside
  LIN {X -9249.921,Y 0.110,Z 34.400,A 89.99666,B 0.00000,C 180.00000} ; preinsert
  LIN {X -9249.921,Y 0.110,Z -215.600,A 89.99666,B 0.00000,C 180.00000} ; insert
  LIN {X -9249.921,Y 0.110,Z -215.600,A 89.99666,B 0.00000,C 180.00000} ; release
  LIN {X -9249.921,Y 0.110,Z 84.400,A 89.99666,B 0.00000,C 180.00000} ; retreat
  ; Step 539, bar 1199
  LIN {X -9124.921,Y 0.110,Z 947.280,A 89.99666,B 0.00000,C 180.00000} ; outside
  LIN {X -9124.921,Y 0.110,Z 34.400,A 89.99666,B 0.00000,C 180.00000} ; preinsert
  LIN {X -9124.921,Y 0.110,Z -215.600,A 89.99666,B 0.00000,C 180.00000} ; insert
  LIN {X -9124.921,Y 0.110,Z -215.600,A 89.99666,B 0.00000,C 180.00000} ; release
  LIN {X -9124.921,Y 0.110,Z 84.400,A 89.99666,B 0.00000,C 180.00000} ; retreat
  ; Step 540, bar 1201
  LIN {X -9015.921,Y 0.110,Z 947.280,A 89.99666,B 0.00000,C 180.00000} ; outside
  LIN {X -9015.921,Y 0.110,Z 34.400,A 89.99666,B 0.00000,C 180.00000} ; preinsert
  LIN {X -9015.921,Y 0.110,Z -215.600,A 89.99666,B 0.00000,C 180.00000} ; insert
  LIN {X -9015.921,Y 0.110,Z -215.600,A 89.99666,B 0.00000,C 180.00000} ; release
  LIN {X -9015.921,Y 0.110,Z 84.400,A 89.99666,B 0.00000,C 180.00000} ; retreat
  ; Step 541, bar 1200
  LIN {X -8999.921,Y 0.110,Z 947.280,A 89.99666,B 0.00000,C 180.00000} ; outside
  LIN {X -8999.921,Y 0.110,Z 34.400,A 89.99666,B 0.00000,C 180.00000} ; preinsert
  LIN {X -8999.921,Y 0.110,Z -215.600,A 89.99666,B 0.00000,C 180.00000} ; insert
  LIN {X -8999.921,Y 0.110,Z -215.600,A 89.99666,B 0.00000,C 180.00000} ; release
  LIN {X -8999.921,Y 0.110,Z 84.400,A 89.99666,B 0.00000,C 180.00000} ; retreat
  ; Step 542, bar 1198
  LIN {X -8874.921,Y 0.110,Z 947.280,A 89.99666,B 0.00000,C 180.00000} ; outside
  LIN {X -8874.921,Y 0.110,Z 34.400,A 89.99666,B 0.00000,C 180.00000} ; preinsert
  LIN {X -8874.921,Y 0.110,Z -215.600,A 89.99666,B 0.00000,C 180.00000} ; insert
  LIN {X -8874.921,Y 0.110,Z -215.600,A 89.99666,B 0.00000,C 180.00000} ; release
  LIN {X -8874.921,Y 0.110,Z 84.400,A 89.99666,B 0.00000,C 180.00000} ; retreat
  ; Step 543, bar 1197
  LIN {X -8749.921,Y 0.110,Z 947.280,A 89.99666,B 0.00000,C 180.00000} ; outside
  LIN {X -8749.921,Y 0.110,Z 34.400,A 89.99666,B 0.00000,C 180.00000} ; preinsert
  LIN {X -8749.921,Y 0.110,Z -215.600,A 89.99666,B 0.00000,C 180.00000} ; insert
  LIN {X -8749.921,Y 0.110,Z -215.600,A 89.99666,B 0.00000,C 180.00000} ; release
  LIN {X -8749.921,Y 0.110,Z 84.400,A 89.99666,B 0.00000,C 180.00000} ; retreat
  ; Step 544, bar 1194
  LIN {X -8624.921,Y 0.110,Z 947.280,A 89.99666,B 0.00000,C 180.00000} ; outside
  LIN {X -8624.921,Y 0.110,Z 34.400,A 89.99666,B 0.00000,C 180.00000} ; preinsert
  LIN {X -8624.921,Y 0.110,Z -215.600,A 89.99666,B 0.00000,C 180.00000} ; insert
  LIN {X -8624.921,Y 0.110,Z -215.600,A 89.99666,B 0.00000,C 180.00000} ; release
  LIN {X -8624.921,Y 0.110,Z 84.400,A 89.99666,B 0.00000,C 180.00000} ; retreat
  ; Step 545, bar 1196
  LIN {X -8515.921,Y 0.110,Z 947.280,A 89.99666,B 0.00000,C 180.00000} ; outside
  LIN {X -8515.921,Y 0.110,Z 34.400,A 89.99666,B 0.00000,C 180.00000} ; preinsert
  LIN {X -8515.921,Y 0.110,Z -215.600,A 89.99666,B 0.00000,C 180.00000} ; insert
  LIN {X -8515.921,Y 0.110,Z -215.600,A 89.99666,B 0.00000,C 180.00000} ; release
  LIN {X -8515.921,Y 0.110,Z 84.400,A 89.99666,B 0.00000,C 180.00000} ; retreat
  ; Step 546, bar 1195
  LIN {X -8499.921,Y 0.110,Z 947.280,A 89.99666,B 0.00000,C 180.00000} ; outside
  LIN {X -8499.921,Y 0.110,Z 34.400,A 89.99666,B 0.00000,C 180.00000} ; preinsert
  LIN {X -8499.921,Y 0.110,Z -215.600,A 89.99666,B 0.00000,C 180.00000} ; insert
  LIN {X -8499.921,Y 0.110,Z -215.600,A 89.99666,B 0.00000,C 180.00000} ; release
  LIN {X -8499.921,Y 0.110,Z 84.400,A 89.99666,B 0.00000,C 180.00000} ; retreat
  ; Step 547, bar 1193
  LIN {X -8374.921,Y 0.110,Z 947.280,A 89.99666,B 0.00000,C 180.00000} ; outside
  LIN {X -8374.921,Y 0.110,Z 34.400,A 89.99666,B 0.00000,C 180.00000} ; preinsert
  LIN {X -8374.921,Y 0.110,Z -215.600,A 89.99666,B 0.00000,C 180.00000} ; insert
  LIN {X -8374.921,Y 0.110,Z -215.600,A 89.99666,B 0.00000,C 180.00000} ; release
  LIN {X -8374.921,Y 0.110,Z 84.400,A 89.99666,B 0.00000,C 180.00000} ; retreat
  ; Step 548, bar 1192
  LIN {X -8249.921,Y 0.110,Z 947.280,A 89.99666,B 0.00000,C 180.00000} ; outside
  LIN {X -8249.921,Y 0.110,Z 34.400,A 89.99666,B 0.00000,C 180.00000} ; preinsert
  LIN {X -8249.921,Y 0.110,Z -215.600,A 89.99666,B 0.00000,C 180.00000} ; insert
  LIN {X -8249.921,Y 0.110,Z -215.600,A 89.99666,B 0.00000,C 180.00000} ; release
  LIN {X -8249.921,Y 0.110,Z 84.400,A 89.99666,B 0.00000,C 180.00000} ; retreat
  ; Step 549, bar 1189
  LIN {X -8124.921,Y 0.110,Z 947.280,A 89.99666,B 0.00000,C 180.00000} ; outside
  LIN {X -8124.921,Y 0.110,Z 34.400,A 89.99666,B 0.00000,C 180.00000} ; preinsert
  LIN {X -8124.921,Y 0.110,Z -215.600,A 89.99666,B 0.00000,C 180.00000} ; insert
  LIN {X -8124.921,Y 0.110,Z -215.600,A 89.99666,B 0.00000,C 180.00000} ; release
  LIN {X -8124.921,Y 0.110,Z 84.400,A 89.99666,B 0.00000,C 180.00000} ; retreat
  ; Step 550, bar 1191
  LIN {X -8015.921,Y 0.110,Z 947.280,A 89.99666,B 0.00000,C 180.00000} ; outside
  LIN {X -8015.921,Y 0.110,Z 34.400,A 89.99666,B 0.00000,C 180.00000} ; preinsert
  LIN {X -8015.921,Y 0.110,Z -215.600,A 89.99666,B 0.00000,C 180.00000} ; insert
  LIN {X -8015.921,Y 0.110,Z -215.600,A 89.99666,B 0.00000,C 180.00000} ; release
  LIN {X -8015.921,Y 0.110,Z 84.400,A 89.99666,B 0.00000,C 180.00000} ; retreat
  ; Step 551, bar 1190
  LIN {X -7999.921,Y 0.110,Z 947.280,A 89.99666,B 0.00000,C 180.00000} ; outside
  LIN {X -7999.921,Y 0.110,Z 34.400,A 89.99666,B 0.00000,C 180.00000} ; preinsert
  LIN {X -7999.921,Y 0.110,Z -215.600,A 89.99666,B 0.00000,C 180.00000} ; insert
  LIN {X -7999.921,Y 0.110,Z -215.600,A 89.99666,B 0.00000,C 180.00000} ; release
  LIN {X -7999.921,Y 0.110,Z 84.400,A 89.99666,B 0.00000,C 180.00000} ; retreat
  ; Step 552, bar 1188
  LIN {X -7874.921,Y 0.110,Z 947.280,A 89.99666,B 0.00000,C 180.00000} ; outside
  LIN {X -7874.921,Y 0.110,Z 34.400,A 89.99666,B 0.00000,C 180.00000} ; preinsert
  LIN {X -7874.921,Y 0.110,Z -215.600,A 89.99666,B 0.00000,C 180.00000} ; insert
  LIN {X -7874.921,Y 0.110,Z -215.600,A 89.99666,B 0.00000,C 180.00000} ; release
  LIN {X -7874.921,Y 0.110,Z 84.400,A 89.99666,B 0.00000,C 180.00000} ; retreat
  ; Step 553, bar 1187
  LIN {X -7749.921,Y 0.110,Z 947.280,A 89.99666,B 0.00000,C 180.00000} ; outside
  LIN {X -7749.921,Y 0.110,Z 34.400,A 89.99666,B 0.00000,C 180.00000} ; preinsert
  LIN {X -7749.921,Y 0.110,Z -215.600,A 89.99666,B 0.00000,C 180.00000} ; insert
  LIN {X -7749.921,Y 0.110,Z -215.600,A 89.99666,B 0.00000,C 180.00000} ; release
  LIN {X -7749.921,Y 0.110,Z 84.400,A 89.99666,B 0.00000,C 180.00000} ; retreat
  ; Step 554, bar 1184
  LIN {X -7624.921,Y 0.110,Z 947.280,A 89.99666,B 0.00000,C 180.00000} ; outside
  LIN {X -7624.921,Y 0.110,Z 34.400,A 89.99666,B 0.00000,C 180.00000} ; preinsert
  LIN {X -7624.921,Y 0.110,Z -215.600,A 89.99666,B 0.00000,C 180.00000} ; insert
  LIN {X -7624.921,Y 0.110,Z -215.600,A 89.99666,B 0.00000,C 180.00000} ; release
  LIN {X -7624.921,Y 0.110,Z 84.400,A 89.99666,B 0.00000,C 180.00000} ; retreat
  ; Step 555, bar 1186
  LIN {X -7515.921,Y 0.110,Z 947.280,A 89.99666,B 0.00000,C 180.00000} ; outside
  LIN {X -7515.921,Y 0.110,Z 34.400,A 89.99666,B 0.00000,C 180.00000} ; preinsert
  LIN {X -7515.921,Y 0.110,Z -215.600,A 89.99666,B 0.00000,C 180.00000} ; insert
  LIN {X -7515.921,Y 0.110,Z -215.600,A 89.99666,B 0.00000,C 180.00000} ; release
  LIN {X -7515.921,Y 0.110,Z 84.400,A 89.99666,B 0.00000,C 180.00000} ; retreat
  ; Step 556, bar 1185
  LIN {X -7499.921,Y 0.110,Z 947.280,A 89.99666,B 0.00000,C 180.00000} ; outside
  LIN {X -7499.921,Y 0.110,Z 34.400,A 89.99666,B 0.00000,C 180.00000} ; preinsert
  LIN {X -7499.921,Y 0.110,Z -215.600,A 89.99666,B 0.00000,C 180.00000} ; insert
  LIN {X -7499.921,Y 0.110,Z -215.600,A 89.99666,B 0.00000,C 180.00000} ; release
  LIN {X -7499.921,Y 0.110,Z 84.400,A 89.99666,B 0.00000,C 180.00000} ; retreat
  ; Step 557, bar 1183
  LIN {X -7374.921,Y 0.110,Z 947.280,A 89.99666,B 0.00000,C 180.00000} ; outside
  LIN {X -7374.921,Y 0.110,Z 34.400,A 89.99666,B 0.00000,C 180.00000} ; preinsert
  LIN {X -7374.921,Y 0.110,Z -215.600,A 89.99666,B 0.00000,C 180.00000} ; insert
  LIN {X -7374.921,Y 0.110,Z -215.600,A 89.99666,B 0.00000,C 180.00000} ; release
  LIN {X -7374.921,Y 0.110,Z 84.400,A 89.99666,B 0.00000,C 180.00000} ; retreat
  ; Step 558, bar 1182
  LIN {X -7249.921,Y 0.110,Z 947.280,A 89.99666,B 0.00000,C 180.00000} ; outside
  LIN {X -7249.921,Y 0.110,Z 34.400,A 89.99666,B 0.00000,C 180.00000} ; preinsert
  LIN {X -7249.921,Y 0.110,Z -215.600,A 89.99666,B 0.00000,C 180.00000} ; insert
  LIN {X -7249.921,Y 0.110,Z -215.600,A 89.99666,B 0.00000,C 180.00000} ; release
  LIN {X -7249.921,Y 0.110,Z 84.400,A 89.99666,B 0.00000,C 180.00000} ; retreat
  ; Step 559, bar 1179
  LIN {X -7124.921,Y 0.110,Z 947.280,A 89.99666,B 0.00000,C 180.00000} ; outside
  LIN {X -7124.921,Y 0.110,Z 34.400,A 89.99666,B 0.00000,C 180.00000} ; preinsert
  LIN {X -7124.921,Y 0.110,Z -215.600,A 89.99666,B 0.00000,C 180.00000} ; insert
  LIN {X -7124.921,Y 0.110,Z -215.600,A 89.99666,B 0.00000,C 180.00000} ; release
  LIN {X -7124.921,Y 0.110,Z 84.400,A 89.99666,B 0.00000,C 180.00000} ; retreat
  ; Step 560, bar 1181
  LIN {X -7015.921,Y 0.110,Z 947.280,A 89.99666,B 0.00000,C 180.00000} ; outside
  LIN {X -7015.921,Y 0.110,Z 34.400,A 89.99666,B 0.00000,C 180.00000} ; preinsert
  LIN {X -7015.921,Y 0.110,Z -215.600,A 89.99666,B 0.00000,C 180.00000} ; insert
  LIN {X -7015.921,Y 0.110,Z -215.600,A 89.99666,B 0.00000,C 180.00000} ; release
  LIN {X -7015.921,Y 0.110,Z 84.400,A 89.99666,B 0.00000,C 180.00000} ; retreat
  ; Step 561, bar 1180
  LIN {X -6999.921,Y 0.110,Z 947.280,A 89.99666,B 0.00000,C 180.00000} ; outside
  LIN {X -6999.921,Y 0.110,Z 34.400,A 89.99666,B 0.00000,C 180.00000} ; preinsert
  LIN {X -6999.921,Y 0.110,Z -215.600,A 89.99666,B 0.00000,C 180.00000} ; insert
  LIN {X -6999.921,Y 0.110,Z -215.600,A 89.99666,B 0.00000,C 180.00000} ; release
  LIN {X -6999.921,Y 0.110,Z 84.400,A 89.99666,B 0.00000,C 180.00000} ; retreat
  ; Step 562, bar 1178
  LIN {X -6874.921,Y 0.110,Z 947.280,A 89.99666,B 0.00000,C 180.00000} ; outside
  LIN {X -6874.921,Y 0.110,Z 34.400,A 89.99666,B 0.00000,C 180.00000} ; preinsert
  LIN {X -6874.921,Y 0.110,Z -215.600,A 89.99666,B 0.00000,C 180.00000} ; insert
  LIN {X -6874.921,Y 0.110,Z -215.600,A 89.99666,B 0.00000,C 180.00000} ; release
  LIN {X -6874.921,Y 0.110,Z 84.400,A 89.99666,B 0.00000,C 180.00000} ; retreat
  ; Step 563, bar 1177
  LIN {X -6749.921,Y 0.110,Z 947.280,A 89.99666,B 0.00000,C 180.00000} ; outside
  LIN {X -6749.921,Y 0.110,Z 34.400,A 89.99666,B 0.00000,C 180.00000} ; preinsert
  LIN {X -6749.921,Y 0.110,Z -215.600,A 89.99666,B 0.00000,C 180.00000} ; insert
  LIN {X -6749.921,Y 0.110,Z -215.600,A 89.99666,B 0.00000,C 180.00000} ; release
  LIN {X -6749.921,Y 0.110,Z 84.400,A 89.99666,B 0.00000,C 180.00000} ; retreat
  ; Step 564, bar 1174
  LIN {X -6624.921,Y 0.110,Z 947.280,A 89.99666,B 0.00000,C 180.00000} ; outside
  LIN {X -6624.921,Y 0.110,Z 34.400,A 89.99666,B 0.00000,C 180.00000} ; preinsert
  LIN {X -6624.921,Y 0.110,Z -215.600,A 89.99666,B 0.00000,C 180.00000} ; insert
  LIN {X -6624.921,Y 0.110,Z -215.600,A 89.99666,B 0.00000,C 180.00000} ; release
  LIN {X -6624.921,Y 0.110,Z 84.400,A 89.99666,B 0.00000,C 180.00000} ; retreat
  ; Step 565, bar 1176
  LIN {X -6515.921,Y 0.110,Z 947.280,A 89.99666,B 0.00000,C 180.00000} ; outside
  LIN {X -6515.921,Y 0.110,Z 34.400,A 89.99666,B 0.00000,C 180.00000} ; preinsert
  LIN {X -6515.921,Y 0.110,Z -215.600,A 89.99666,B 0.00000,C 180.00000} ; insert
  LIN {X -6515.921,Y 0.110,Z -215.600,A 89.99666,B 0.00000,C 180.00000} ; release
  LIN {X -6515.921,Y 0.110,Z 84.400,A 89.99666,B 0.00000,C 180.00000} ; retreat
  ; Step 566, bar 1175
  LIN {X -6499.921,Y 0.110,Z 947.280,A 89.99666,B 0.00000,C 180.00000} ; outside
  LIN {X -6499.921,Y 0.110,Z 34.400,A 89.99666,B 0.00000,C 180.00000} ; preinsert
  LIN {X -6499.921,Y 0.110,Z -215.600,A 89.99666,B 0.00000,C 180.00000} ; insert
  LIN {X -6499.921,Y 0.110,Z -215.600,A 89.99666,B 0.00000,C 180.00000} ; release
  LIN {X -6499.921,Y 0.110,Z 84.400,A 89.99666,B 0.00000,C 180.00000} ; retreat
  ; Step 567, bar 1173
  LIN {X -6374.921,Y 0.110,Z 947.280,A 89.99666,B 0.00000,C 180.00000} ; outside
  LIN {X -6374.921,Y 0.110,Z 34.400,A 89.99666,B 0.00000,C 180.00000} ; preinsert
  LIN {X -6374.921,Y 0.110,Z -215.600,A 89.99666,B 0.00000,C 180.00000} ; insert
  LIN {X -6374.921,Y 0.110,Z -215.600,A 89.99666,B 0.00000,C 180.00000} ; release
  LIN {X -6374.921,Y 0.110,Z 84.400,A 89.99666,B 0.00000,C 180.00000} ; retreat
  ; Step 568, bar 1172
  LIN {X -6249.921,Y 0.110,Z 947.280,A 89.99666,B 0.00000,C 180.00000} ; outside
  LIN {X -6249.921,Y 0.110,Z 34.400,A 89.99666,B 0.00000,C 180.00000} ; preinsert
  LIN {X -6249.921,Y 0.110,Z -215.600,A 89.99666,B 0.00000,C 180.00000} ; insert
  LIN {X -6249.921,Y 0.110,Z -215.600,A 89.99666,B 0.00000,C 180.00000} ; release
  LIN {X -6249.921,Y 0.110,Z 84.400,A 89.99666,B 0.00000,C 180.00000} ; retreat
  ; Step 569, bar 1169
  LIN {X -6124.921,Y 0.110,Z 947.280,A 89.99666,B 0.00000,C 180.00000} ; outside
  LIN {X -6124.921,Y 0.110,Z 34.400,A 89.99666,B 0.00000,C 180.00000} ; preinsert
  LIN {X -6124.921,Y 0.110,Z -215.600,A 89.99666,B 0.00000,C 180.00000} ; insert
  LIN {X -6124.921,Y 0.110,Z -215.600,A 89.99666,B 0.00000,C 180.00000} ; release
  LIN {X -6124.921,Y 0.110,Z 84.400,A 89.99666,B 0.00000,C 180.00000} ; retreat
  ; Step 570, bar 1168
  LIN {X -5999.921,Y 0.110,Z 947.280,A 89.99666,B 0.00000,C 180.00000} ; outside
  LIN {X -5999.921,Y 0.110,Z 34.400,A 89.99666,B 0.00000,C 180.00000} ; preinsert
  LIN {X -5999.921,Y 0.110,Z -215.600,A 89.99666,B 0.00000,C 180.00000} ; insert
  LIN {X -5999.921,Y 0.110,Z -215.600,A 89.99666,B 0.00000,C 180.00000} ; release
  LIN {X -5999.921,Y 0.110,Z 84.400,A 89.99666,B 0.00000,C 180.00000} ; retreat
  ; Step 571, bar 1171
  LIN {X -5890.921,Y 0.110,Z 947.280,A 89.99666,B 0.00000,C 180.00000} ; outside
  LIN {X -5890.921,Y 0.110,Z 34.400,A 89.99666,B 0.00000,C 180.00000} ; preinsert
  LIN {X -5890.921,Y 0.110,Z -215.600,A 89.99666,B 0.00000,C 180.00000} ; insert
  LIN {X -5890.921,Y 0.110,Z -215.600,A 89.99666,B 0.00000,C 180.00000} ; release
  LIN {X -5890.921,Y 0.110,Z 84.400,A 89.99666,B 0.00000,C 180.00000} ; retreat
  ; Step 572, bar 1170
  LIN {X -5874.921,Y 0.110,Z 947.280,A 89.99666,B 0.00000,C 180.00000} ; outside
  LIN {X -5874.921,Y 0.110,Z 34.400,A 89.99666,B 0.00000,C 180.00000} ; preinsert
  LIN {X -5874.921,Y 0.110,Z -215.600,A 89.99666,B 0.00000,C 180.00000} ; insert
  LIN {X -5874.921,Y 0.110,Z -215.600,A 89.99666,B 0.00000,C 180.00000} ; release
  LIN {X -5874.921,Y 0.110,Z 84.400,A 89.99666,B 0.00000,C 180.00000} ; retreat
  ; Step 573, bar 1167
  LIN {X -5749.921,Y 0.110,Z 947.280,A 89.99666,B 0.00000,C 180.00000} ; outside
  LIN {X -5749.921,Y 0.110,Z 34.400,A 89.99666,B 0.00000,C 180.00000} ; preinsert
  LIN {X -5749.921,Y 0.110,Z -215.600,A 89.99666,B 0.00000,C 180.00000} ; insert
  LIN {X -5749.921,Y 0.110,Z -215.600,A 89.99666,B 0.00000,C 180.00000} ; release
  LIN {X -5749.921,Y 0.110,Z 84.400,A 89.99666,B 0.00000,C 180.00000} ; retreat
  ; Step 574, bar 1164
  LIN {X -5624.921,Y 0.110,Z 947.280,A 89.99666,B 0.00000,C 180.00000} ; outside
  LIN {X -5624.921,Y 0.110,Z 34.400,A 89.99666,B 0.00000,C 180.00000} ; preinsert
  LIN {X -5624.921,Y 0.110,Z -215.600,A 89.99666,B 0.00000,C 180.00000} ; insert
  LIN {X -5624.921,Y 0.110,Z -215.600,A 89.99666,B 0.00000,C 180.00000} ; release
  LIN {X -5624.921,Y 0.110,Z 84.400,A 89.99666,B 0.00000,C 180.00000} ; retreat
  ; Step 575, bar 1166
  LIN {X -5515.921,Y 0.110,Z 947.280,A 89.99666,B 0.00000,C 180.00000} ; outside
  LIN {X -5515.921,Y 0.110,Z 34.400,A 89.99666,B 0.00000,C 180.00000} ; preinsert
  LIN {X -5515.921,Y 0.110,Z -215.600,A 89.99666,B 0.00000,C 180.00000} ; insert
  LIN {X -5515.921,Y 0.110,Z -215.600,A 89.99666,B 0.00000,C 180.00000} ; release
  LIN {X -5515.921,Y 0.110,Z 84.400,A 89.99666,B 0.00000,C 180.00000} ; retreat
  ; Step 576, bar 1165
  LIN {X -5499.921,Y 0.110,Z 947.280,A 89.99666,B 0.00000,C 180.00000} ; outside
  LIN {X -5499.921,Y 0.110,Z 34.400,A 89.99666,B 0.00000,C 180.00000} ; preinsert
  LIN {X -5499.921,Y 0.110,Z -215.600,A 89.99666,B 0.00000,C 180.00000} ; insert
  LIN {X -5499.921,Y 0.110,Z -215.600,A 89.99666,B 0.00000,C 180.00000} ; release
  LIN {X -5499.921,Y 0.110,Z 84.400,A 89.99666,B 0.00000,C 180.00000} ; retreat
  ; Step 577, bar 1163
  LIN {X -5374.921,Y 0.110,Z 947.280,A 89.99666,B 0.00000,C 180.00000} ; outside
  LIN {X -5374.921,Y 0.110,Z 34.400,A 89.99666,B 0.00000,C 180.00000} ; preinsert
  LIN {X -5374.921,Y 0.110,Z -215.600,A 89.99666,B 0.00000,C 180.00000} ; insert
  LIN {X -5374.921,Y 0.110,Z -215.600,A 89.99666,B 0.00000,C 180.00000} ; release
  LIN {X -5374.921,Y 0.110,Z 84.400,A 89.99666,B 0.00000,C 180.00000} ; retreat
  ; Step 578, bar 1162
  LIN {X -5249.921,Y 0.110,Z 947.280,A 89.99666,B 0.00000,C 180.00000} ; outside
  LIN {X -5249.921,Y 0.110,Z 34.400,A 89.99666,B 0.00000,C 180.00000} ; preinsert
  LIN {X -5249.921,Y 0.110,Z -215.600,A 89.99666,B 0.00000,C 180.00000} ; insert
  LIN {X -5249.921,Y 0.110,Z -215.600,A 89.99666,B 0.00000,C 180.00000} ; release
  LIN {X -5249.921,Y 0.110,Z 84.400,A 89.99666,B 0.00000,C 180.00000} ; retreat
  ; Step 579, bar 1159
  LIN {X -5124.921,Y 0.110,Z 947.280,A 89.99666,B 0.00000,C 180.00000} ; outside
  LIN {X -5124.921,Y 0.110,Z 34.400,A 89.99666,B 0.00000,C 180.00000} ; preinsert
  LIN {X -5124.921,Y 0.110,Z -215.600,A 89.99666,B 0.00000,C 180.00000} ; insert
  LIN {X -5124.921,Y 0.110,Z -215.600,A 89.99666,B 0.00000,C 180.00000} ; release
  LIN {X -5124.921,Y 0.110,Z 84.400,A 89.99666,B 0.00000,C 180.00000} ; retreat
  ; Step 580, bar 1161
  LIN {X -5015.921,Y 0.110,Z 947.280,A 89.99666,B 0.00000,C 180.00000} ; outside
  LIN {X -5015.921,Y 0.110,Z 34.400,A 89.99666,B 0.00000,C 180.00000} ; preinsert
  LIN {X -5015.921,Y 0.110,Z -215.600,A 89.99666,B 0.00000,C 180.00000} ; insert
  LIN {X -5015.921,Y 0.110,Z -215.600,A 89.99666,B 0.00000,C 180.00000} ; release
  LIN {X -5015.921,Y 0.110,Z 84.400,A 89.99666,B 0.00000,C 180.00000} ; retreat
  ; Step 581, bar 1160
  LIN {X -4999.921,Y 0.110,Z 947.280,A 89.99666,B 0.00000,C 180.00000} ; outside
  LIN {X -4999.921,Y 0.110,Z 34.400,A 89.99666,B 0.00000,C 180.00000} ; preinsert
  LIN {X -4999.921,Y 0.110,Z -215.600,A 89.99666,B 0.00000,C 180.00000} ; insert
  LIN {X -4999.921,Y 0.110,Z -215.600,A 89.99666,B 0.00000,C 180.00000} ; release
  LIN {X -4999.921,Y 0.110,Z 84.400,A 89.99666,B 0.00000,C 180.00000} ; retreat
  ; Step 582, bar 1158
  LIN {X -4874.921,Y 0.110,Z 947.280,A 89.99666,B 0.00000,C 180.00000} ; outside
  LIN {X -4874.921,Y 0.110,Z 34.400,A 89.99666,B 0.00000,C 180.00000} ; preinsert
  LIN {X -4874.921,Y 0.110,Z -215.600,A 89.99666,B 0.00000,C 180.00000} ; insert
  LIN {X -4874.921,Y 0.110,Z -215.600,A 89.99666,B 0.00000,C 180.00000} ; release
  LIN {X -4874.921,Y 0.110,Z 84.400,A 89.99666,B 0.00000,C 180.00000} ; retreat
  ; Step 583, bar 1157
  LIN {X -4749.921,Y 0.110,Z 947.280,A 89.99666,B 0.00000,C 180.00000} ; outside
  LIN {X -4749.921,Y 0.110,Z 34.400,A 89.99666,B 0.00000,C 180.00000} ; preinsert
  LIN {X -4749.921,Y 0.110,Z -215.600,A 89.99666,B 0.00000,C 180.00000} ; insert
  LIN {X -4749.921,Y 0.110,Z -215.600,A 89.99666,B 0.00000,C 180.00000} ; release
  LIN {X -4749.921,Y 0.110,Z 84.400,A 89.99666,B 0.00000,C 180.00000} ; retreat
  ; Step 584, bar 1154
  LIN {X -4624.921,Y 0.110,Z 947.280,A 89.99666,B 0.00000,C 180.00000} ; outside
  LIN {X -4624.921,Y 0.110,Z 34.400,A 89.99666,B 0.00000,C 180.00000} ; preinsert
  LIN {X -4624.921,Y 0.110,Z -215.600,A 89.99666,B 0.00000,C 180.00000} ; insert
  LIN {X -4624.921,Y 0.110,Z -215.600,A 89.99666,B 0.00000,C 180.00000} ; release
  LIN {X -4624.921,Y 0.110,Z 84.400,A 89.99666,B 0.00000,C 180.00000} ; retreat
  ; Step 585, bar 1156
  LIN {X -4515.921,Y 0.110,Z 947.280,A 89.99666,B 0.00000,C 180.00000} ; outside
  LIN {X -4515.921,Y 0.110,Z 34.400,A 89.99666,B 0.00000,C 180.00000} ; preinsert
  LIN {X -4515.921,Y 0.110,Z -215.600,A 89.99666,B 0.00000,C 180.00000} ; insert
  LIN {X -4515.921,Y 0.110,Z -215.600,A 89.99666,B 0.00000,C 180.00000} ; release
  LIN {X -4515.921,Y 0.110,Z 84.400,A 89.99666,B 0.00000,C 180.00000} ; retreat
  ; Step 586, bar 1155
  LIN {X -4499.921,Y 0.110,Z 947.280,A 89.99666,B 0.00000,C 180.00000} ; outside
  LIN {X -4499.921,Y 0.110,Z 34.400,A 89.99666,B 0.00000,C 180.00000} ; preinsert
  LIN {X -4499.921,Y 0.110,Z -215.600,A 89.99666,B 0.00000,C 180.00000} ; insert
  LIN {X -4499.921,Y 0.110,Z -215.600,A 89.99666,B 0.00000,C 180.00000} ; release
  LIN {X -4499.921,Y 0.110,Z 84.400,A 89.99666,B 0.00000,C 180.00000} ; retreat
  ; Step 587, bar 1153
  LIN {X -4374.921,Y 0.110,Z 947.280,A 89.99666,B 0.00000,C 180.00000} ; outside
  LIN {X -4374.921,Y 0.110,Z 34.400,A 89.99666,B 0.00000,C 180.00000} ; preinsert
  LIN {X -4374.921,Y 0.110,Z -215.600,A 89.99666,B 0.00000,C 180.00000} ; insert
  LIN {X -4374.921,Y 0.110,Z -215.600,A 89.99666,B 0.00000,C 180.00000} ; release
  LIN {X -4374.921,Y 0.110,Z 84.400,A 89.99666,B 0.00000,C 180.00000} ; retreat
  ; Step 588, bar 1152
  LIN {X -4249.921,Y 0.110,Z 947.280,A 89.99666,B 0.00000,C 180.00000} ; outside
  LIN {X -4249.921,Y 0.110,Z 34.400,A 89.99666,B 0.00000,C 180.00000} ; preinsert
  LIN {X -4249.921,Y 0.110,Z -215.600,A 89.99666,B 0.00000,C 180.00000} ; insert
  LIN {X -4249.921,Y 0.110,Z -215.600,A 89.99666,B 0.00000,C 180.00000} ; release
  LIN {X -4249.921,Y 0.110,Z 84.400,A 89.99666,B 0.00000,C 180.00000} ; retreat
  ; Step 589, bar 1149
  LIN {X -4124.921,Y 0.110,Z 947.280,A 89.99666,B 0.00000,C 180.00000} ; outside
  LIN {X -4124.921,Y 0.110,Z 34.400,A 89.99666,B 0.00000,C 180.00000} ; preinsert
  LIN {X -4124.921,Y 0.110,Z -215.600,A 89.99666,B 0.00000,C 180.00000} ; insert
  LIN {X -4124.921,Y 0.110,Z -215.600,A 89.99666,B 0.00000,C 180.00000} ; release
  LIN {X -4124.921,Y 0.110,Z 84.400,A 89.99666,B 0.00000,C 180.00000} ; retreat
  ; Step 590, bar 1151
  LIN {X -4015.921,Y 0.110,Z 947.280,A 89.99666,B 0.00000,C 180.00000} ; outside
  LIN {X -4015.921,Y 0.110,Z 34.400,A 89.99666,B 0.00000,C 180.00000} ; preinsert
  LIN {X -4015.921,Y 0.110,Z -215.600,A 89.99666,B 0.00000,C 180.00000} ; insert
  LIN {X -4015.921,Y 0.110,Z -215.600,A 89.99666,B 0.00000,C 180.00000} ; release
  LIN {X -4015.921,Y 0.110,Z 84.400,A 89.99666,B 0.00000,C 180.00000} ; retreat
  ; Step 591, bar 1150
  LIN {X -3999.921,Y 0.110,Z 947.280,A 89.99666,B 0.00000,C 180.00000} ; outside
  LIN {X -3999.921,Y 0.110,Z 34.400,A 89.99666,B 0.00000,C 180.00000} ; preinsert
  LIN {X -3999.921,Y 0.110,Z -215.600,A 89.99666,B 0.00000,C 180.00000} ; insert
  LIN {X -3999.921,Y 0.110,Z -215.600,A 89.99666,B 0.00000,C 180.00000} ; release
  LIN {X -3999.921,Y 0.110,Z 84.400,A 89.99666,B 0.00000,C 180.00000} ; retreat
  ; Step 592, bar 1148
  LIN {X -3874.921,Y 0.110,Z 947.280,A 89.99666,B 0.00000,C 180.00000} ; outside
  LIN {X -3874.921,Y 0.110,Z 34.400,A 89.99666,B 0.00000,C 180.00000} ; preinsert
  LIN {X -3874.921,Y 0.110,Z -215.600,A 89.99666,B 0.00000,C 180.00000} ; insert
  LIN {X -3874.921,Y 0.110,Z -215.600,A 89.99666,B 0.00000,C 180.00000} ; release
  LIN {X -3874.921,Y 0.110,Z 84.400,A 89.99666,B 0.00000,C 180.00000} ; retreat
  ; Step 593, bar 1147
  LIN {X -3749.921,Y 0.110,Z 947.280,A 89.99666,B 0.00000,C 180.00000} ; outside
  LIN {X -3749.921,Y 0.110,Z 34.400,A 89.99666,B 0.00000,C 180.00000} ; preinsert
  LIN {X -3749.921,Y 0.110,Z -215.600,A 89.99666,B 0.00000,C 180.00000} ; insert
  LIN {X -3749.921,Y 0.110,Z -215.600,A 89.99666,B 0.00000,C 180.00000} ; release
  LIN {X -3749.921,Y 0.110,Z 84.400,A 89.99666,B 0.00000,C 180.00000} ; retreat
  ; Step 594, bar 1144
  LIN {X -3624.921,Y 0.110,Z 947.280,A 89.99666,B 0.00000,C 180.00000} ; outside
  LIN {X -3624.921,Y 0.110,Z 34.400,A 89.99666,B 0.00000,C 180.00000} ; preinsert
  LIN {X -3624.921,Y 0.110,Z -215.600,A 89.99666,B 0.00000,C 180.00000} ; insert
  LIN {X -3624.921,Y 0.110,Z -215.600,A 89.99666,B 0.00000,C 180.00000} ; release
  LIN {X -3624.921,Y 0.110,Z 84.400,A 89.99666,B 0.00000,C 180.00000} ; retreat
  ; Step 595, bar 1146
  LIN {X -3515.921,Y 0.110,Z 947.280,A 89.99666,B 0.00000,C 180.00000} ; outside
  LIN {X -3515.921,Y 0.110,Z 34.400,A 89.99666,B 0.00000,C 180.00000} ; preinsert
  LIN {X -3515.921,Y 0.110,Z -215.600,A 89.99666,B 0.00000,C 180.00000} ; insert
  LIN {X -3515.921,Y 0.110,Z -215.600,A 89.99666,B 0.00000,C 180.00000} ; release
  LIN {X -3515.921,Y 0.110,Z 84.400,A 89.99666,B 0.00000,C 180.00000} ; retreat
  ; Step 596, bar 1145
  LIN {X -3499.921,Y 0.110,Z 947.280,A 89.99666,B 0.00000,C 180.00000} ; outside
  LIN {X -3499.921,Y 0.110,Z 34.400,A 89.99666,B 0.00000,C 180.00000} ; preinsert
  LIN {X -3499.921,Y 0.110,Z -215.600,A 89.99666,B 0.00000,C 180.00000} ; insert
  LIN {X -3499.921,Y 0.110,Z -215.600,A 89.99666,B 0.00000,C 180.00000} ; release
  LIN {X -3499.921,Y 0.110,Z 84.400,A 89.99666,B 0.00000,C 180.00000} ; retreat
  ; Step 597, bar 1143
  LIN {X -3374.921,Y 0.110,Z 947.280,A 89.99666,B 0.00000,C 180.00000} ; outside
  LIN {X -3374.921,Y 0.110,Z 34.400,A 89.99666,B 0.00000,C 180.00000} ; preinsert
  LIN {X -3374.921,Y 0.110,Z -215.600,A 89.99666,B 0.00000,C 180.00000} ; insert
  LIN {X -3374.921,Y 0.110,Z -215.600,A 89.99666,B 0.00000,C 180.00000} ; release
  LIN {X -3374.921,Y 0.110,Z 84.400,A 89.99666,B 0.00000,C 180.00000} ; retreat
  ; Step 598, bar 1142
  LIN {X -3249.921,Y 0.110,Z 947.280,A 89.99666,B 0.00000,C 180.00000} ; outside
  LIN {X -3249.921,Y 0.110,Z 34.400,A 89.99666,B 0.00000,C 180.00000} ; preinsert
  LIN {X -3249.921,Y 0.110,Z -215.600,A 89.99666,B 0.00000,C 180.00000} ; insert
  LIN {X -3249.921,Y 0.110,Z -215.600,A 89.99666,B 0.00000,C 180.00000} ; release
  LIN {X -3249.921,Y 0.110,Z 84.400,A 89.99666,B 0.00000,C 180.00000} ; retreat
  ; Step 599, bar 1139
  LIN {X -3124.921,Y 0.110,Z 947.280,A 89.99666,B 0.00000,C 180.00000} ; outside
  LIN {X -3124.921,Y 0.110,Z 34.400,A 89.99666,B 0.00000,C 180.00000} ; preinsert
  LIN {X -3124.921,Y 0.110,Z -215.600,A 89.99666,B 0.00000,C 180.00000} ; insert
  LIN {X -3124.921,Y 0.110,Z -215.600,A 89.99666,B 0.00000,C 180.00000} ; release
  LIN {X -3124.921,Y 0.110,Z 84.400,A 89.99666,B 0.00000,C 180.00000} ; retreat
  ; Step 600, bar 1141
  LIN {X -3015.921,Y 0.110,Z 947.280,A 89.99666,B 0.00000,C 180.00000} ; outside
  LIN {X -3015.921,Y 0.110,Z 34.400,A 89.99666,B 0.00000,C 180.00000} ; preinsert
  LIN {X -3015.921,Y 0.110,Z -215.600,A 89.99666,B 0.00000,C 180.00000} ; insert
  LIN {X -3015.921,Y 0.110,Z -215.600,A 89.99666,B 0.00000,C 180.00000} ; release
  LIN {X -3015.921,Y 0.110,Z 84.400,A 89.99666,B 0.00000,C 180.00000} ; retreat
  ; Step 601, bar 1140
  LIN {X -2999.921,Y 0.110,Z 947.280,A 89.99666,B 0.00000,C 180.00000} ; outside
  LIN {X -2999.921,Y 0.110,Z 34.400,A 89.99666,B 0.00000,C 180.00000} ; preinsert
  LIN {X -2999.921,Y 0.110,Z -215.600,A 89.99666,B 0.00000,C 180.00000} ; insert
  LIN {X -2999.921,Y 0.110,Z -215.600,A 89.99666,B 0.00000,C 180.00000} ; release
  LIN {X -2999.921,Y 0.110,Z 84.400,A 89.99666,B 0.00000,C 180.00000} ; retreat
  ; Step 602, bar 1138
  LIN {X -2874.921,Y 0.110,Z 947.280,A 89.99666,B 0.00000,C 180.00000} ; outside
  LIN {X -2874.921,Y 0.110,Z 34.400,A 89.99666,B 0.00000,C 180.00000} ; preinsert
  LIN {X -2874.921,Y 0.110,Z -215.600,A 89.99666,B 0.00000,C 180.00000} ; insert
  LIN {X -2874.921,Y 0.110,Z -215.600,A 89.99666,B 0.00000,C 180.00000} ; release
  LIN {X -2874.921,Y 0.110,Z 84.400,A 89.99666,B 0.00000,C 180.00000} ; retreat
  ; Step 603, bar 1137
  LIN {X -2749.921,Y 0.110,Z 947.280,A 89.99666,B 0.00000,C 180.00000} ; outside
  LIN {X -2749.921,Y 0.110,Z 34.400,A 89.99666,B 0.00000,C 180.00000} ; preinsert
  LIN {X -2749.921,Y 0.110,Z -215.600,A 89.99666,B 0.00000,C 180.00000} ; insert
  LIN {X -2749.921,Y 0.110,Z -215.600,A 89.99666,B 0.00000,C 180.00000} ; release
  LIN {X -2749.921,Y 0.110,Z 84.400,A 89.99666,B 0.00000,C 180.00000} ; retreat
  ; Step 604, bar 1134
  LIN {X -2624.921,Y 0.110,Z 947.280,A 89.99666,B 0.00000,C 180.00000} ; outside
  LIN {X -2624.921,Y 0.110,Z 34.400,A 89.99666,B 0.00000,C 180.00000} ; preinsert
  LIN {X -2624.921,Y 0.110,Z -215.600,A 89.99666,B 0.00000,C 180.00000} ; insert
  LIN {X -2624.921,Y 0.110,Z -215.600,A 89.99666,B 0.00000,C 180.00000} ; release
  LIN {X -2624.921,Y 0.110,Z 84.400,A 89.99666,B 0.00000,C 180.00000} ; retreat
  ; Step 605, bar 1136
  LIN {X -2515.921,Y 0.110,Z 947.280,A 89.99666,B 0.00000,C 180.00000} ; outside
  LIN {X -2515.921,Y 0.110,Z 34.400,A 89.99666,B 0.00000,C 180.00000} ; preinsert
  LIN {X -2515.921,Y 0.110,Z -215.600,A 89.99666,B 0.00000,C 180.00000} ; insert
  LIN {X -2515.921,Y 0.110,Z -215.600,A 89.99666,B 0.00000,C 180.00000} ; release
  LIN {X -2515.921,Y 0.110,Z 84.400,A 89.99666,B 0.00000,C 180.00000} ; retreat
  ; Step 606, bar 1135
  LIN {X -2499.921,Y 0.110,Z 947.280,A 89.99666,B 0.00000,C 180.00000} ; outside
  LIN {X -2499.921,Y 0.110,Z 34.400,A 89.99666,B 0.00000,C 180.00000} ; preinsert
  LIN {X -2499.921,Y 0.110,Z -215.600,A 89.99666,B 0.00000,C 180.00000} ; insert
  LIN {X -2499.921,Y 0.110,Z -215.600,A 89.99666,B 0.00000,C 180.00000} ; release
  LIN {X -2499.921,Y 0.110,Z 84.400,A 89.99666,B 0.00000,C 180.00000} ; retreat
  ; Step 607, bar 1133
  LIN {X -2374.921,Y 0.110,Z 947.280,A 89.99666,B 0.00000,C 180.00000} ; outside
  LIN {X -2374.921,Y 0.110,Z 34.400,A 89.99666,B 0.00000,C 180.00000} ; preinsert
  LIN {X -2374.921,Y 0.110,Z -215.600,A 89.99666,B 0.00000,C 180.00000} ; insert
  LIN {X -2374.921,Y 0.110,Z -215.600,A 89.99666,B 0.00000,C 180.00000} ; release
  LIN {X -2374.921,Y 0.110,Z 84.400,A 89.99666,B 0.00000,C 180.00000} ; retreat
  ; Step 608, bar 1132
  LIN {X -2249.921,Y 0.110,Z 947.280,A 89.99666,B 0.00000,C 180.00000} ; outside
  LIN {X -2249.921,Y 0.110,Z 34.400,A 89.99666,B 0.00000,C 180.00000} ; preinsert
  LIN {X -2249.921,Y 0.110,Z -215.600,A 89.99666,B 0.00000,C 180.00000} ; insert
  LIN {X -2249.921,Y 0.110,Z -215.600,A 89.99666,B 0.00000,C 180.00000} ; release
  LIN {X -2249.921,Y 0.110,Z 84.400,A 89.99666,B 0.00000,C 180.00000} ; retreat
  ; Step 609, bar 1129
  LIN {X -2124.921,Y 0.110,Z 947.280,A 89.99666,B 0.00000,C 180.00000} ; outside
  LIN {X -2124.921,Y 0.110,Z 34.400,A 89.99666,B 0.00000,C 180.00000} ; preinsert
  LIN {X -2124.921,Y 0.110,Z -215.600,A 89.99666,B 0.00000,C 180.00000} ; insert
  LIN {X -2124.921,Y 0.110,Z -215.600,A 89.99666,B 0.00000,C 180.00000} ; release
  LIN {X -2124.921,Y 0.110,Z 84.400,A 89.99666,B 0.00000,C 180.00000} ; retreat
  ; Step 610, bar 1128
  LIN {X -1999.921,Y 0.110,Z 947.280,A 89.99666,B 0.00000,C 180.00000} ; outside
  LIN {X -1999.921,Y 0.110,Z 34.400,A 89.99666,B 0.00000,C 180.00000} ; preinsert
  LIN {X -1999.921,Y 0.110,Z -215.600,A 89.99666,B 0.00000,C 180.00000} ; insert
  LIN {X -1999.921,Y 0.110,Z -215.600,A 89.99666,B 0.00000,C 180.00000} ; release
  LIN {X -1999.921,Y 0.110,Z 84.400,A 89.99666,B 0.00000,C 180.00000} ; retreat
  ; Step 611, bar 1131
  LIN {X -1890.921,Y 0.110,Z 947.280,A 89.99666,B 0.00000,C 180.00000} ; outside
  LIN {X -1890.921,Y 0.110,Z 34.400,A 89.99666,B 0.00000,C 180.00000} ; preinsert
  LIN {X -1890.921,Y 0.110,Z -215.600,A 89.99666,B 0.00000,C 180.00000} ; insert
  LIN {X -1890.921,Y 0.110,Z -215.600,A 89.99666,B 0.00000,C 180.00000} ; release
  LIN {X -1890.921,Y 0.110,Z 84.400,A 89.99666,B 0.00000,C 180.00000} ; retreat
  ; Step 612, bar 1130
  LIN {X -1874.921,Y 0.110,Z 947.280,A 89.99666,B 0.00000,C 180.00000} ; outside
  LIN {X -1874.921,Y 0.110,Z 34.400,A 89.99666,B 0.00000,C 180.00000} ; preinsert
  LIN {X -1874.921,Y 0.110,Z -215.600,A 89.99666,B 0.00000,C 180.00000} ; insert
  LIN {X -1874.921,Y 0.110,Z -215.600,A 89.99666,B 0.00000,C 180.00000} ; release
  LIN {X -1874.921,Y 0.110,Z 84.400,A 89.99666,B 0.00000,C 180.00000} ; retreat
  ; Step 613, bar 1127
  LIN {X -1749.921,Y 0.110,Z 947.280,A 89.99666,B 0.00000,C 180.00000} ; outside
  LIN {X -1749.921,Y 0.110,Z 34.400,A 89.99666,B 0.00000,C 180.00000} ; preinsert
  LIN {X -1749.921,Y 0.110,Z -215.600,A 89.99666,B 0.00000,C 180.00000} ; insert
  LIN {X -1749.921,Y 0.110,Z -215.600,A 89.99666,B 0.00000,C 180.00000} ; release
  LIN {X -1749.921,Y 0.110,Z 84.400,A 89.99666,B 0.00000,C 180.00000} ; retreat
  ; Step 614, bar 1124
  LIN {X -1624.921,Y 0.110,Z 947.280,A 89.99666,B 0.00000,C 180.00000} ; outside
  LIN {X -1624.921,Y 0.110,Z 34.400,A 89.99666,B 0.00000,C 180.00000} ; preinsert
  LIN {X -1624.921,Y 0.110,Z -215.600,A 89.99666,B 0.00000,C 180.00000} ; insert
  LIN {X -1624.921,Y 0.110,Z -215.600,A 89.99666,B 0.00000,C 180.00000} ; release
  LIN {X -1624.921,Y 0.110,Z 84.400,A 89.99666,B 0.00000,C 180.00000} ; retreat
  ; Step 615, bar 1126
  LIN {X -1515.921,Y 0.110,Z 947.280,A 89.99666,B 0.00000,C 180.00000} ; outside
  LIN {X -1515.921,Y 0.110,Z 34.400,A 89.99666,B 0.00000,C 180.00000} ; preinsert
  LIN {X -1515.921,Y 0.110,Z -215.600,A 89.99666,B 0.00000,C 180.00000} ; insert
  LIN {X -1515.921,Y 0.110,Z -215.600,A 89.99666,B 0.00000,C 180.00000} ; release
  LIN {X -1515.921,Y 0.110,Z 84.400,A 89.99666,B 0.00000,C 180.00000} ; retreat
  ; Step 616, bar 1125
  LIN {X -1499.921,Y 0.110,Z 947.280,A 89.99666,B 0.00000,C 180.00000} ; outside
  LIN {X -1499.921,Y 0.110,Z 34.400,A 89.99666,B 0.00000,C 180.00000} ; preinsert
  LIN {X -1499.921,Y 0.110,Z -215.600,A 89.99666,B 0.00000,C 180.00000} ; insert
  LIN {X -1499.921,Y 0.110,Z -215.600,A 89.99666,B 0.00000,C 180.00000} ; release
  LIN {X -1499.921,Y 0.110,Z 84.400,A 89.99666,B 0.00000,C 180.00000} ; retreat
  ; Step 617, bar 1123
  LIN {X -1374.921,Y 0.110,Z 947.280,A 89.99666,B 0.00000,C 180.00000} ; outside
  LIN {X -1374.921,Y 0.110,Z 34.400,A 89.99666,B 0.00000,C 180.00000} ; preinsert
  LIN {X -1374.921,Y 0.110,Z -215.600,A 89.99666,B 0.00000,C 180.00000} ; insert
  LIN {X -1374.921,Y 0.110,Z -215.600,A 89.99666,B 0.00000,C 180.00000} ; release
  LIN {X -1374.921,Y 0.110,Z 84.400,A 89.99666,B 0.00000,C 180.00000} ; retreat
  ; Step 618, bar 1122
  LIN {X -1249.921,Y 0.110,Z 947.280,A 89.99666,B 0.00000,C 180.00000} ; outside
  LIN {X -1249.921,Y 0.110,Z 34.400,A 89.99666,B 0.00000,C 180.00000} ; preinsert
  LIN {X -1249.921,Y 0.110,Z -215.600,A 89.99666,B 0.00000,C 180.00000} ; insert
  LIN {X -1249.921,Y 0.110,Z -215.600,A 89.99666,B 0.00000,C 180.00000} ; release
  LIN {X -1249.921,Y 0.110,Z 84.400,A 89.99666,B 0.00000,C 180.00000} ; retreat
  ; Step 619, bar 1119
  LIN {X -1124.921,Y 0.110,Z 947.280,A 89.99666,B 0.00000,C 180.00000} ; outside
  LIN {X -1124.921,Y 0.110,Z 34.400,A 89.99666,B 0.00000,C 180.00000} ; preinsert
  LIN {X -1124.921,Y 0.110,Z -215.600,A 89.99666,B 0.00000,C 180.00000} ; insert
  LIN {X -1124.921,Y 0.110,Z -215.600,A 89.99666,B 0.00000,C 180.00000} ; release
  LIN {X -1124.921,Y 0.110,Z 84.400,A 89.99666,B 0.00000,C 180.00000} ; retreat
  ; Step 620, bar 1121
  LIN {X -1015.921,Y 0.110,Z 947.280,A 89.99666,B 0.00000,C 180.00000} ; outside
  LIN {X -1015.921,Y 0.110,Z 34.400,A 89.99666,B 0.00000,C 180.00000} ; preinsert
  LIN {X -1015.921,Y 0.110,Z -215.600,A 89.99666,B 0.00000,C 180.00000} ; insert
  LIN {X -1015.921,Y 0.110,Z -215.600,A 89.99666,B 0.00000,C 180.00000} ; release
  LIN {X -1015.921,Y 0.110,Z 84.400,A 89.99666,B 0.00000,C 180.00000} ; retreat
  ; Step 621, bar 1120
  LIN {X -999.921,Y 0.110,Z 947.280,A 89.99666,B 0.00000,C 180.00000} ; outside
  LIN {X -999.921,Y 0.110,Z 34.400,A 89.99666,B 0.00000,C 180.00000} ; preinsert
  LIN {X -999.921,Y 0.110,Z -215.600,A 89.99666,B 0.00000,C 180.00000} ; insert
  LIN {X -999.921,Y 0.110,Z -215.600,A 89.99666,B 0.00000,C 180.00000} ; release
  LIN {X -999.921,Y 0.110,Z 84.400,A 89.99666,B 0.00000,C 180.00000} ; retreat
  ; Step 622, bar 1118
  LIN {X -874.921,Y 0.110,Z 947.280,A 89.99666,B 0.00000,C 180.00000} ; outside
  LIN {X -874.921,Y 0.110,Z 34.400,A 89.99666,B 0.00000,C 180.00000} ; preinsert
  LIN {X -874.921,Y 0.110,Z -215.600,A 89.99666,B 0.00000,C 180.00000} ; insert
  LIN {X -874.921,Y 0.110,Z -215.600,A 89.99666,B 0.00000,C 180.00000} ; release
  LIN {X -874.921,Y 0.110,Z 84.400,A 89.99666,B 0.00000,C 180.00000} ; retreat
  ; Step 623, bar 1117
  LIN {X -749.921,Y 0.110,Z 947.280,A 89.99666,B 0.00000,C 180.00000} ; outside
  LIN {X -749.921,Y 0.110,Z 34.400,A 89.99666,B 0.00000,C 180.00000} ; preinsert
  LIN {X -749.921,Y 0.110,Z -215.600,A 89.99666,B 0.00000,C 180.00000} ; insert
  LIN {X -749.921,Y 0.110,Z -215.600,A 89.99666,B 0.00000,C 180.00000} ; release
  LIN {X -749.921,Y 0.110,Z 84.400,A 89.99666,B 0.00000,C 180.00000} ; retreat
  ; Step 624, bar 1114
  LIN {X -624.921,Y 0.110,Z 947.280,A 89.99666,B 0.00000,C 180.00000} ; outside
  LIN {X -624.921,Y 0.110,Z 34.400,A 89.99666,B 0.00000,C 180.00000} ; preinsert
  LIN {X -624.921,Y 0.110,Z -215.600,A 89.99666,B 0.00000,C 180.00000} ; insert
  LIN {X -624.921,Y 0.110,Z -215.600,A 89.99666,B 0.00000,C 180.00000} ; release
  LIN {X -624.921,Y 0.110,Z 84.400,A 89.99666,B 0.00000,C 180.00000} ; retreat
  ; Step 625, bar 1116
  LIN {X -515.921,Y 0.110,Z 947.280,A 89.99666,B 0.00000,C 180.00000} ; outside
  LIN {X -515.921,Y 0.110,Z 34.400,A 89.99666,B 0.00000,C 180.00000} ; preinsert
  LIN {X -515.921,Y 0.110,Z -215.600,A 89.99666,B 0.00000,C 180.00000} ; insert
  LIN {X -515.921,Y 0.110,Z -215.600,A 89.99666,B 0.00000,C 180.00000} ; release
  LIN {X -515.921,Y 0.110,Z 84.400,A 89.99666,B 0.00000,C 180.00000} ; retreat
  ; Step 626, bar 1115
  LIN {X -499.921,Y 0.110,Z 947.280,A 89.99666,B 0.00000,C 180.00000} ; outside
  LIN {X -499.921,Y 0.110,Z 34.400,A 89.99666,B 0.00000,C 180.00000} ; preinsert
  LIN {X -499.921,Y 0.110,Z -215.600,A 89.99666,B 0.00000,C 180.00000} ; insert
  LIN {X -499.921,Y 0.110,Z -215.600,A 89.99666,B 0.00000,C 180.00000} ; release
  LIN {X -499.921,Y 0.110,Z 84.400,A 89.99666,B 0.00000,C 180.00000} ; retreat
  ; Step 627, bar 1113
  LIN {X -374.921,Y 0.110,Z 947.280,A 89.99666,B 0.00000,C 180.00000} ; outside
  LIN {X -374.921,Y 0.110,Z 34.400,A 89.99666,B 0.00000,C 180.00000} ; preinsert
  LIN {X -374.921,Y 0.110,Z -215.600,A 89.99666,B 0.00000,C 180.00000} ; insert
  LIN {X -374.921,Y 0.110,Z -215.600,A 89.99666,B 0.00000,C 180.00000} ; release
  LIN {X -374.921,Y 0.110,Z 84.400,A 89.99666,B 0.00000,C 180.00000} ; retreat
  ; Step 628, bar 1112
  LIN {X -249.921,Y 0.110,Z 947.280,A 89.99666,B 0.00000,C 180.00000} ; outside
  LIN {X -249.921,Y 0.110,Z 34.400,A 89.99666,B 0.00000,C 180.00000} ; preinsert
  LIN {X -249.921,Y 0.110,Z -215.600,A 89.99666,B 0.00000,C 180.00000} ; insert
  LIN {X -249.921,Y 0.110,Z -215.600,A 89.99666,B 0.00000,C 180.00000} ; release
  LIN {X -249.921,Y 0.110,Z 84.400,A 89.99666,B 0.00000,C 180.00000} ; retreat
  ; Step 629, bar 1111
  LIN {X -124.921,Y 0.110,Z 947.280,A 89.99666,B 0.00000,C 180.00000} ; outside
  LIN {X -124.921,Y 0.110,Z 34.400,A 89.99666,B 0.00000,C 180.00000} ; preinsert
  LIN {X -124.921,Y 0.110,Z -215.600,A 89.99666,B 0.00000,C 180.00000} ; insert
  LIN {X -124.921,Y 0.110,Z -215.600,A 89.99666,B 0.00000,C 180.00000} ; release
  LIN {X -124.921,Y 0.110,Z 84.400,A 89.99666,B 0.00000,C 180.00000} ; retreat
  ; Step 630, bar 894
  LIN {X -0.079,Y 0.097,Z 947.280,A 90.00334,B 0.00000,C 180.00000} ; outside
  LIN {X -0.079,Y 0.097,Z 34.400,A 90.00334,B 0.00000,C 180.00000} ; preinsert
  LIN {X -0.079,Y 0.097,Z -215.600,A 90.00334,B 0.00000,C 180.00000} ; insert
  LIN {X -0.079,Y 0.097,Z -215.600,A 90.00334,B 0.00000,C 180.00000} ; release
  LIN {X -0.079,Y 0.097,Z 84.400,A 90.00334,B 0.00000,C 180.00000} ; retreat
  ; Step 631, bar 895
  LIN {X 15.921,Y 0.097,Z 947.280,A 90.00334,B 0.00000,C 180.00000} ; outside
  LIN {X 15.921,Y 0.097,Z 34.400,A 90.00334,B 0.00000,C 180.00000} ; preinsert
  LIN {X 15.921,Y 0.097,Z -215.600,A 90.00334,B 0.00000,C 180.00000} ; insert
  LIN {X 15.921,Y 0.097,Z -215.600,A 90.00334,B 0.00000,C 180.00000} ; release
  LIN {X 15.921,Y 0.097,Z 84.400,A 90.00334,B 0.00000,C 180.00000} ; retreat
  ; Step 632, bar 892
  LIN {X 124.921,Y 0.097,Z 947.280,A 90.00334,B 0.00000,C 180.00000} ; outside
  LIN {X 124.921,Y 0.097,Z 34.400,A 90.00334,B 0.00000,C 180.00000} ; preinsert
  LIN {X 124.921,Y 0.097,Z -215.600,A 90.00334,B 0.00000,C 180.00000} ; insert
  LIN {X 124.921,Y 0.097,Z -215.600,A 90.00334,B 0.00000,C 180.00000} ; release
  LIN {X 124.921,Y 0.097,Z 84.400,A 90.00334,B 0.00000,C 180.00000} ; retreat
  ; Step 633, bar 896
  LIN {X 249.921,Y 0.097,Z 947.280,A 90.00334,B 0.00000,C 180.00000} ; outside
  LIN {X 249.921,Y 0.097,Z 34.400,A 90.00334,B 0.00000,C 180.00000} ; preinsert
  LIN {X 249.921,Y 0.097,Z -215.600,A 90.00334,B 0.00000,C 180.00000} ; insert
  LIN {X 249.921,Y 0.097,Z -215.600,A 90.00334,B 0.00000,C 180.00000} ; release
  LIN {X 249.921,Y 0.097,Z 84.400,A 90.00334,B 0.00000,C 180.00000} ; retreat
  ; Step 634, bar 897
  LIN {X 374.921,Y 0.097,Z 947.280,A 90.00334,B 0.00000,C 180.00000} ; outside
  LIN {X 374.921,Y 0.097,Z 34.400,A 90.00334,B 0.00000,C 180.00000} ; preinsert
  LIN {X 374.921,Y 0.097,Z -215.600,A 90.00334,B 0.00000,C 180.00000} ; insert
  LIN {X 374.921,Y 0.097,Z -215.600,A 90.00334,B 0.00000,C 180.00000} ; release
  LIN {X 374.921,Y 0.097,Z 84.400,A 90.00334,B 0.00000,C 180.00000} ; retreat
  ; Step 635, bar 899
  LIN {X 499.921,Y 0.097,Z 947.280,A 90.00334,B 0.00000,C 180.00000} ; outside
  LIN {X 499.921,Y 0.097,Z 34.400,A 90.00334,B 0.00000,C 180.00000} ; preinsert
  LIN {X 499.921,Y 0.097,Z -215.600,A 90.00334,B 0.00000,C 180.00000} ; insert
  LIN {X 499.921,Y 0.097,Z -215.600,A 90.00334,B 0.00000,C 180.00000} ; release
  LIN {X 499.921,Y 0.097,Z 84.400,A 90.00334,B 0.00000,C 180.00000} ; retreat
  ; Step 636, bar 900
  LIN {X 515.921,Y 0.097,Z 947.280,A 90.00334,B 0.00000,C 180.00000} ; outside
  LIN {X 515.921,Y 0.097,Z 34.400,A 90.00334,B 0.00000,C 180.00000} ; preinsert
  LIN {X 515.921,Y 0.097,Z -215.600,A 90.00334,B 0.00000,C 180.00000} ; insert
  LIN {X 515.921,Y 0.097,Z -215.600,A 90.00334,B 0.00000,C 180.00000} ; release
  LIN {X 515.921,Y 0.097,Z 84.400,A 90.00334,B 0.00000,C 180.00000} ; retreat
  ; Step 637, bar 898
  LIN {X 624.921,Y 0.097,Z 947.280,A 90.00334,B 0.00000,C 180.00000} ; outside
  LIN {X 624.921,Y 0.097,Z 34.400,A 90.00334,B 0.00000,C 180.00000} ; preinsert
  LIN {X 624.921,Y 0.097,Z -215.600,A 90.00334,B 0.00000,C 180.00000} ; insert
  LIN {X 624.921,Y 0.097,Z -215.600,A 90.00334,B 0.00000,C 180.00000} ; release
  LIN {X 624.921,Y 0.097,Z 84.400,A 90.00334,B 0.00000,C 180.00000} ; retreat
  ; Step 638, bar 901
  LIN {X 749.921,Y 0.097,Z 947.280,A 90.00334,B 0.00000,C 180.00000} ; outside
  LIN {X 749.921,Y 0.097,Z 34.400,A 90.00334,B 0.00000,C 180.00000} ; preinsert
  LIN {X 749.921,Y 0.097,Z -215.600,A 90.00334,B 0.00000,C 180.00000} ; insert
  LIN {X 749.921,Y 0.097,Z -215.600,A 90.00334,B 0.00000,C 180.00000} ; release
  LIN {X 749.921,Y 0.097,Z 84.400,A 90.00334,B 0.00000,C 180.00000} ; retreat
  ; Step 639, bar 902
  LIN {X 874.921,Y 0.097,Z 947.280,A 90.00334,B 0.00000,C 180.00000} ; outside
  LIN {X 874.921,Y 0.097,Z 34.400,A 90.00334,B 0.00000,C 180.00000} ; preinsert
  LIN {X 874.921,Y 0.097,Z -215.600,A 90.00334,B 0.00000,C 180.00000} ; insert
  LIN {X 874.921,Y 0.097,Z -215.600,A 90.00334,B 0.00000,C 180.00000} ; release
  LIN {X 874.921,Y 0.097,Z 84.400,A 90.00334,B 0.00000,C 180.00000} ; retreat
  ; Step 640, bar 904
  LIN {X 999.921,Y 0.097,Z 947.280,A 90.00334,B 0.00000,C 180.00000} ; outside
  LIN {X 999.921,Y 0.097,Z 34.400,A 90.00334,B 0.00000,C 180.00000} ; preinsert
  LIN {X 999.921,Y 0.097,Z -215.600,A 90.00334,B 0.00000,C 180.00000} ; insert
  LIN {X 999.921,Y 0.097,Z -215.600,A 90.00334,B 0.00000,C 180.00000} ; release
  LIN {X 999.921,Y 0.097,Z 84.400,A 90.00334,B 0.00000,C 180.00000} ; retreat
  ; Step 641, bar 905
  LIN {X 1015.921,Y 0.097,Z 947.280,A 90.00334,B 0.00000,C 180.00000} ; outside
  LIN {X 1015.921,Y 0.097,Z 34.400,A 90.00334,B 0.00000,C 180.00000} ; preinsert
  LIN {X 1015.921,Y 0.097,Z -215.600,A 90.00334,B 0.00000,C 180.00000} ; insert
  LIN {X 1015.921,Y 0.097,Z -215.600,A 90.00334,B 0.00000,C 180.00000} ; release
  LIN {X 1015.921,Y 0.097,Z 84.400,A 90.00334,B 0.00000,C 180.00000} ; retreat
  ; Step 642, bar 903
  LIN {X 1124.921,Y 0.097,Z 947.280,A 90.00334,B 0.00000,C 180.00000} ; outside
  LIN {X 1124.921,Y 0.097,Z 34.400,A 90.00334,B 0.00000,C 180.00000} ; preinsert
  LIN {X 1124.921,Y 0.097,Z -215.600,A 90.00334,B 0.00000,C 180.00000} ; insert
  LIN {X 1124.921,Y 0.097,Z -215.600,A 90.00334,B 0.00000,C 180.00000} ; release
  LIN {X 1124.921,Y 0.097,Z 84.400,A 90.00334,B 0.00000,C 180.00000} ; retreat
  ; Step 643, bar 906
  LIN {X 1249.921,Y 0.097,Z 947.280,A 90.00334,B 0.00000,C 180.00000} ; outside
  LIN {X 1249.921,Y 0.097,Z 34.400,A 90.00334,B 0.00000,C 180.00000} ; preinsert
  LIN {X 1249.921,Y 0.097,Z -215.600,A 90.00334,B 0.00000,C 180.00000} ; insert
  LIN {X 1249.921,Y 0.097,Z -215.600,A 90.00334,B 0.00000,C 180.00000} ; release
  LIN {X 1249.921,Y 0.097,Z 84.400,A 90.00334,B 0.00000,C 180.00000} ; retreat
  ; Step 644, bar 907
  LIN {X 1374.921,Y 0.097,Z 947.280,A 90.00334,B 0.00000,C 180.00000} ; outside
  LIN {X 1374.921,Y 0.097,Z 34.400,A 90.00334,B 0.00000,C 180.00000} ; preinsert
  LIN {X 1374.921,Y 0.097,Z -215.600,A 90.00334,B 0.00000,C 180.00000} ; insert
  LIN {X 1374.921,Y 0.097,Z -215.600,A 90.00334,B 0.00000,C 180.00000} ; release
  LIN {X 1374.921,Y 0.097,Z 84.400,A 90.00334,B 0.00000,C 180.00000} ; retreat
  ; Step 645, bar 909
  LIN {X 1499.921,Y 0.097,Z 947.280,A 90.00334,B 0.00000,C 180.00000} ; outside
  LIN {X 1499.921,Y 0.097,Z 34.400,A 90.00334,B 0.00000,C 180.00000} ; preinsert
  LIN {X 1499.921,Y 0.097,Z -215.600,A 90.00334,B 0.00000,C 180.00000} ; insert
  LIN {X 1499.921,Y 0.097,Z -215.600,A 90.00334,B 0.00000,C 180.00000} ; release
  LIN {X 1499.921,Y 0.097,Z 84.400,A 90.00334,B 0.00000,C 180.00000} ; retreat
  ; Step 646, bar 910
  LIN {X 1515.921,Y 0.097,Z 947.280,A 90.00334,B 0.00000,C 180.00000} ; outside
  LIN {X 1515.921,Y 0.097,Z 34.400,A 90.00334,B 0.00000,C 180.00000} ; preinsert
  LIN {X 1515.921,Y 0.097,Z -215.600,A 90.00334,B 0.00000,C 180.00000} ; insert
  LIN {X 1515.921,Y 0.097,Z -215.600,A 90.00334,B 0.00000,C 180.00000} ; release
  LIN {X 1515.921,Y 0.097,Z 84.400,A 90.00334,B 0.00000,C 180.00000} ; retreat
  ; Step 647, bar 908
  LIN {X 1624.921,Y 0.097,Z 947.280,A 90.00334,B 0.00000,C 180.00000} ; outside
  LIN {X 1624.921,Y 0.097,Z 34.400,A 90.00334,B 0.00000,C 180.00000} ; preinsert
  LIN {X 1624.921,Y 0.097,Z -215.600,A 90.00334,B 0.00000,C 180.00000} ; insert
  LIN {X 1624.921,Y 0.097,Z -215.600,A 90.00334,B 0.00000,C 180.00000} ; release
  LIN {X 1624.921,Y 0.097,Z 84.400,A 90.00334,B 0.00000,C 180.00000} ; retreat
  ; Step 648, bar 911
  LIN {X 1749.921,Y 0.097,Z 947.280,A 90.00334,B 0.00000,C 180.00000} ; outside
  LIN {X 1749.921,Y 0.097,Z 34.400,A 90.00334,B 0.00000,C 180.00000} ; preinsert
  LIN {X 1749.921,Y 0.097,Z -215.600,A 90.00334,B 0.00000,C 180.00000} ; insert
  LIN {X 1749.921,Y 0.097,Z -215.600,A 90.00334,B 0.00000,C 180.00000} ; release
  LIN {X 1749.921,Y 0.097,Z 84.400,A 90.00334,B 0.00000,C 180.00000} ; retreat
  ; Step 649, bar 914
  LIN {X 1874.921,Y 0.097,Z 947.280,A 90.00334,B 0.00000,C 180.00000} ; outside
  LIN {X 1874.921,Y 0.097,Z 34.400,A 90.00334,B 0.00000,C 180.00000} ; preinsert
  LIN {X 1874.921,Y 0.097,Z -215.600,A 90.00334,B 0.00000,C 180.00000} ; insert
  LIN {X 1874.921,Y 0.097,Z -215.600,A 90.00334,B 0.00000,C 180.00000} ; release
  LIN {X 1874.921,Y 0.097,Z 84.400,A 90.00334,B 0.00000,C 180.00000} ; retreat
  ; Step 650, bar 915
  LIN {X 1890.921,Y 0.097,Z 947.280,A 90.00334,B 0.00000,C 180.00000} ; outside
  LIN {X 1890.921,Y 0.097,Z 34.400,A 90.00334,B 0.00000,C 180.00000} ; preinsert
  LIN {X 1890.921,Y 0.097,Z -215.600,A 90.00334,B 0.00000,C 180.00000} ; insert
  LIN {X 1890.921,Y 0.097,Z -215.600,A 90.00334,B 0.00000,C 180.00000} ; release
  LIN {X 1890.921,Y 0.097,Z 84.400,A 90.00334,B 0.00000,C 180.00000} ; retreat
  ; Step 651, bar 912
  LIN {X 1999.921,Y 0.097,Z 947.280,A 90.00334,B 0.00000,C 180.00000} ; outside
  LIN {X 1999.921,Y 0.097,Z 34.400,A 90.00334,B 0.00000,C 180.00000} ; preinsert
  LIN {X 1999.921,Y 0.097,Z -215.600,A 90.00334,B 0.00000,C 180.00000} ; insert
  LIN {X 1999.921,Y 0.097,Z -215.600,A 90.00334,B 0.00000,C 180.00000} ; release
  LIN {X 1999.921,Y 0.097,Z 84.400,A 90.00334,B 0.00000,C 180.00000} ; retreat
  ; Step 652, bar 913
  LIN {X 2124.921,Y 0.097,Z 947.280,A 90.00334,B 0.00000,C 180.00000} ; outside
  LIN {X 2124.921,Y 0.097,Z 34.400,A 90.00334,B 0.00000,C 180.00000} ; preinsert
  LIN {X 2124.921,Y 0.097,Z -215.600,A 90.00334,B 0.00000,C 180.00000} ; insert
  LIN {X 2124.921,Y 0.097,Z -215.600,A 90.00334,B 0.00000,C 180.00000} ; release
  LIN {X 2124.921,Y 0.097,Z 84.400,A 90.00334,B 0.00000,C 180.00000} ; retreat
  ; Step 653, bar 916
  LIN {X 2249.921,Y 0.097,Z 947.280,A 90.00334,B 0.00000,C 180.00000} ; outside
  LIN {X 2249.921,Y 0.097,Z 34.400,A 90.00334,B 0.00000,C 180.00000} ; preinsert
  LIN {X 2249.921,Y 0.097,Z -215.600,A 90.00334,B 0.00000,C 180.00000} ; insert
  LIN {X 2249.921,Y 0.097,Z -215.600,A 90.00334,B 0.00000,C 180.00000} ; release
  LIN {X 2249.921,Y 0.097,Z 84.400,A 90.00334,B 0.00000,C 180.00000} ; retreat
  ; Step 654, bar 917
  LIN {X 2374.921,Y 0.097,Z 947.280,A 90.00334,B 0.00000,C 180.00000} ; outside
  LIN {X 2374.921,Y 0.097,Z 34.400,A 90.00334,B 0.00000,C 180.00000} ; preinsert
  LIN {X 2374.921,Y 0.097,Z -215.600,A 90.00334,B 0.00000,C 180.00000} ; insert
  LIN {X 2374.921,Y 0.097,Z -215.600,A 90.00334,B 0.00000,C 180.00000} ; release
  LIN {X 2374.921,Y 0.097,Z 84.400,A 90.00334,B 0.00000,C 180.00000} ; retreat
  ; Step 655, bar 919
  LIN {X 2499.921,Y 0.097,Z 947.280,A 90.00334,B 0.00000,C 180.00000} ; outside
  LIN {X 2499.921,Y 0.097,Z 34.400,A 90.00334,B 0.00000,C 180.00000} ; preinsert
  LIN {X 2499.921,Y 0.097,Z -215.600,A 90.00334,B 0.00000,C 180.00000} ; insert
  LIN {X 2499.921,Y 0.097,Z -215.600,A 90.00334,B 0.00000,C 180.00000} ; release
  LIN {X 2499.921,Y 0.097,Z 84.400,A 90.00334,B 0.00000,C 180.00000} ; retreat
  ; Step 656, bar 920
  LIN {X 2515.921,Y 0.097,Z 947.280,A 90.00334,B 0.00000,C 180.00000} ; outside
  LIN {X 2515.921,Y 0.097,Z 34.400,A 90.00334,B 0.00000,C 180.00000} ; preinsert
  LIN {X 2515.921,Y 0.097,Z -215.600,A 90.00334,B 0.00000,C 180.00000} ; insert
  LIN {X 2515.921,Y 0.097,Z -215.600,A 90.00334,B 0.00000,C 180.00000} ; release
  LIN {X 2515.921,Y 0.097,Z 84.400,A 90.00334,B 0.00000,C 180.00000} ; retreat
  ; Step 657, bar 918
  LIN {X 2624.921,Y 0.097,Z 947.280,A 90.00334,B 0.00000,C 180.00000} ; outside
  LIN {X 2624.921,Y 0.097,Z 34.400,A 90.00334,B 0.00000,C 180.00000} ; preinsert
  LIN {X 2624.921,Y 0.097,Z -215.600,A 90.00334,B 0.00000,C 180.00000} ; insert
  LIN {X 2624.921,Y 0.097,Z -215.600,A 90.00334,B 0.00000,C 180.00000} ; release
  LIN {X 2624.921,Y 0.097,Z 84.400,A 90.00334,B 0.00000,C 180.00000} ; retreat
  ; Step 658, bar 921
  LIN {X 2749.921,Y 0.097,Z 947.280,A 90.00334,B 0.00000,C 180.00000} ; outside
  LIN {X 2749.921,Y 0.097,Z 34.400,A 90.00334,B 0.00000,C 180.00000} ; preinsert
  LIN {X 2749.921,Y 0.097,Z -215.600,A 90.00334,B 0.00000,C 180.00000} ; insert
  LIN {X 2749.921,Y 0.097,Z -215.600,A 90.00334,B 0.00000,C 180.00000} ; release
  LIN {X 2749.921,Y 0.097,Z 84.400,A 90.00334,B 0.00000,C 180.00000} ; retreat
  ; Step 659, bar 922
  LIN {X 2874.921,Y 0.097,Z 947.280,A 90.00334,B 0.00000,C 180.00000} ; outside
  LIN {X 2874.921,Y 0.097,Z 34.400,A 90.00334,B 0.00000,C 180.00000} ; preinsert
  LIN {X 2874.921,Y 0.097,Z -215.600,A 90.00334,B 0.00000,C 180.00000} ; insert
  LIN {X 2874.921,Y 0.097,Z -215.600,A 90.00334,B 0.00000,C 180.00000} ; release
  LIN {X 2874.921,Y 0.097,Z 84.400,A 90.00334,B 0.00000,C 180.00000} ; retreat
  ; Step 660, bar 924
  LIN {X 2999.921,Y 0.097,Z 947.280,A 90.00334,B 0.00000,C 180.00000} ; outside
  LIN {X 2999.921,Y 0.097,Z 34.400,A 90.00334,B 0.00000,C 180.00000} ; preinsert
  LIN {X 2999.921,Y 0.097,Z -215.600,A 90.00334,B 0.00000,C 180.00000} ; insert
  LIN {X 2999.921,Y 0.097,Z -215.600,A 90.00334,B 0.00000,C 180.00000} ; release
  LIN {X 2999.921,Y 0.097,Z 84.400,A 90.00334,B 0.00000,C 180.00000} ; retreat
  ; Step 661, bar 925
  LIN {X 3015.921,Y 0.097,Z 947.280,A 90.00334,B 0.00000,C 180.00000} ; outside
  LIN {X 3015.921,Y 0.097,Z 34.400,A 90.00334,B 0.00000,C 180.00000} ; preinsert
  LIN {X 3015.921,Y 0.097,Z -215.600,A 90.00334,B 0.00000,C 180.00000} ; insert
  LIN {X 3015.921,Y 0.097,Z -215.600,A 90.00334,B 0.00000,C 180.00000} ; release
  LIN {X 3015.921,Y 0.097,Z 84.400,A 90.00334,B 0.00000,C 180.00000} ; retreat
  ; Step 662, bar 923
  LIN {X 3124.921,Y 0.097,Z 947.280,A 90.00334,B 0.00000,C 180.00000} ; outside
  LIN {X 3124.921,Y 0.097,Z 34.400,A 90.00334,B 0.00000,C 180.00000} ; preinsert
  LIN {X 3124.921,Y 0.097,Z -215.600,A 90.00334,B 0.00000,C 180.00000} ; insert
  LIN {X 3124.921,Y 0.097,Z -215.600,A 90.00334,B 0.00000,C 180.00000} ; release
  LIN {X 3124.921,Y 0.097,Z 84.400,A 90.00334,B 0.00000,C 180.00000} ; retreat
  ; Step 663, bar 926
  LIN {X 3249.921,Y 0.097,Z 947.280,A 90.00334,B 0.00000,C 180.00000} ; outside
  LIN {X 3249.921,Y 0.097,Z 34.400,A 90.00334,B 0.00000,C 180.00000} ; preinsert
  LIN {X 3249.921,Y 0.097,Z -215.600,A 90.00334,B 0.00000,C 180.00000} ; insert
  LIN {X 3249.921,Y 0.097,Z -215.600,A 90.00334,B 0.00000,C 180.00000} ; release
  LIN {X 3249.921,Y 0.097,Z 84.400,A 90.00334,B 0.00000,C 180.00000} ; retreat
  ; Step 664, bar 927
  LIN {X 3374.921,Y 0.097,Z 947.280,A 90.00334,B 0.00000,C 180.00000} ; outside
  LIN {X 3374.921,Y 0.097,Z 34.400,A 90.00334,B 0.00000,C 180.00000} ; preinsert
  LIN {X 3374.921,Y 0.097,Z -215.600,A 90.00334,B 0.00000,C 180.00000} ; insert
  LIN {X 3374.921,Y 0.097,Z -215.600,A 90.00334,B 0.00000,C 180.00000} ; release
  LIN {X 3374.921,Y 0.097,Z 84.400,A 90.00334,B 0.00000,C 180.00000} ; retreat
  ; Step 665, bar 929
  LIN {X 3499.921,Y 0.097,Z 947.280,A 90.00334,B 0.00000,C 180.00000} ; outside
  LIN {X 3499.921,Y 0.097,Z 34.400,A 90.00334,B 0.00000,C 180.00000} ; preinsert
  LIN {X 3499.921,Y 0.097,Z -215.600,A 90.00334,B 0.00000,C 180.00000} ; insert
  LIN {X 3499.921,Y 0.097,Z -215.600,A 90.00334,B 0.00000,C 180.00000} ; release
  LIN {X 3499.921,Y 0.097,Z 84.400,A 90.00334,B 0.00000,C 180.00000} ; retreat
  ; Step 666, bar 930
  LIN {X 3515.921,Y 0.097,Z 947.280,A 90.00334,B 0.00000,C 180.00000} ; outside
  LIN {X 3515.921,Y 0.097,Z 34.400,A 90.00334,B 0.00000,C 180.00000} ; preinsert
  LIN {X 3515.921,Y 0.097,Z -215.600,A 90.00334,B 0.00000,C 180.00000} ; insert
  LIN {X 3515.921,Y 0.097,Z -215.600,A 90.00334,B 0.00000,C 180.00000} ; release
  LIN {X 3515.921,Y 0.097,Z 84.400,A 90.00334,B 0.00000,C 180.00000} ; retreat
  ; Step 667, bar 928
  LIN {X 3624.921,Y 0.097,Z 947.280,A 90.00334,B 0.00000,C 180.00000} ; outside
  LIN {X 3624.921,Y 0.097,Z 34.400,A 90.00334,B 0.00000,C 180.00000} ; preinsert
  LIN {X 3624.921,Y 0.097,Z -215.600,A 90.00334,B 0.00000,C 180.00000} ; insert
  LIN {X 3624.921,Y 0.097,Z -215.600,A 90.00334,B 0.00000,C 180.00000} ; release
  LIN {X 3624.921,Y 0.097,Z 84.400,A 90.00334,B 0.00000,C 180.00000} ; retreat
  ; Step 668, bar 931
  LIN {X 3749.921,Y 0.097,Z 947.280,A 90.00334,B 0.00000,C 180.00000} ; outside
  LIN {X 3749.921,Y 0.097,Z 34.400,A 90.00334,B 0.00000,C 180.00000} ; preinsert
  LIN {X 3749.921,Y 0.097,Z -215.600,A 90.00334,B 0.00000,C 180.00000} ; insert
  LIN {X 3749.921,Y 0.097,Z -215.600,A 90.00334,B 0.00000,C 180.00000} ; release
  LIN {X 3749.921,Y 0.097,Z 84.400,A 90.00334,B 0.00000,C 180.00000} ; retreat
  ; Step 669, bar 932
  LIN {X 3874.921,Y 0.097,Z 947.280,A 90.00334,B 0.00000,C 180.00000} ; outside
  LIN {X 3874.921,Y 0.097,Z 34.400,A 90.00334,B 0.00000,C 180.00000} ; preinsert
  LIN {X 3874.921,Y 0.097,Z -215.600,A 90.00334,B 0.00000,C 180.00000} ; insert
  LIN {X 3874.921,Y 0.097,Z -215.600,A 90.00334,B 0.00000,C 180.00000} ; release
  LIN {X 3874.921,Y 0.097,Z 84.400,A 90.00334,B 0.00000,C 180.00000} ; retreat
  ; Step 670, bar 934
  LIN {X 3999.921,Y 0.097,Z 947.280,A 90.00334,B 0.00000,C 180.00000} ; outside
  LIN {X 3999.921,Y 0.097,Z 34.400,A 90.00334,B 0.00000,C 180.00000} ; preinsert
  LIN {X 3999.921,Y 0.097,Z -215.600,A 90.00334,B 0.00000,C 180.00000} ; insert
  LIN {X 3999.921,Y 0.097,Z -215.600,A 90.00334,B 0.00000,C 180.00000} ; release
  LIN {X 3999.921,Y 0.097,Z 84.400,A 90.00334,B 0.00000,C 180.00000} ; retreat
  ; Step 671, bar 935
  LIN {X 4015.921,Y 0.097,Z 947.280,A 90.00334,B 0.00000,C 180.00000} ; outside
  LIN {X 4015.921,Y 0.097,Z 34.400,A 90.00334,B 0.00000,C 180.00000} ; preinsert
  LIN {X 4015.921,Y 0.097,Z -215.600,A 90.00334,B 0.00000,C 180.00000} ; insert
  LIN {X 4015.921,Y 0.097,Z -215.600,A 90.00334,B 0.00000,C 180.00000} ; release
  LIN {X 4015.921,Y 0.097,Z 84.400,A 90.00334,B 0.00000,C 180.00000} ; retreat
  ; Step 672, bar 933
  LIN {X 4124.921,Y 0.097,Z 947.280,A 90.00334,B 0.00000,C 180.00000} ; outside
  LIN {X 4124.921,Y 0.097,Z 34.400,A 90.00334,B 0.00000,C 180.00000} ; preinsert
  LIN {X 4124.921,Y 0.097,Z -215.600,A 90.00334,B 0.00000,C 180.00000} ; insert
  LIN {X 4124.921,Y 0.097,Z -215.600,A 90.00334,B 0.00000,C 180.00000} ; release
  LIN {X 4124.921,Y 0.097,Z 84.400,A 90.00334,B 0.00000,C 180.00000} ; retreat
  ; Step 673, bar 936
  LIN {X 4249.921,Y 0.097,Z 947.280,A 90.00334,B 0.00000,C 180.00000} ; outside
  LIN {X 4249.921,Y 0.097,Z 34.400,A 90.00334,B 0.00000,C 180.00000} ; preinsert
  LIN {X 4249.921,Y 0.097,Z -215.600,A 90.00334,B 0.00000,C 180.00000} ; insert
  LIN {X 4249.921,Y 0.097,Z -215.600,A 90.00334,B 0.00000,C 180.00000} ; release
  LIN {X 4249.921,Y 0.097,Z 84.400,A 90.00334,B 0.00000,C 180.00000} ; retreat
  ; Step 674, bar 937
  LIN {X 4374.921,Y 0.097,Z 947.280,A 90.00334,B 0.00000,C 180.00000} ; outside
  LIN {X 4374.921,Y 0.097,Z 34.400,A 90.00334,B 0.00000,C 180.00000} ; preinsert
  LIN {X 4374.921,Y 0.097,Z -215.600,A 90.00334,B 0.00000,C 180.00000} ; insert
  LIN {X 4374.921,Y 0.097,Z -215.600,A 90.00334,B 0.00000,C 180.00000} ; release
  LIN {X 4374.921,Y 0.097,Z 84.400,A 90.00334,B 0.00000,C 180.00000} ; retreat
  ; Step 675, bar 939
  LIN {X 4499.921,Y 0.097,Z 947.280,A 90.00334,B 0.00000,C 180.00000} ; outside
  LIN {X 4499.921,Y 0.097,Z 34.400,A 90.00334,B 0.00000,C 180.00000} ; preinsert
  LIN {X 4499.921,Y 0.097,Z -215.600,A 90.00334,B 0.00000,C 180.00000} ; insert
  LIN {X 4499.921,Y 0.097,Z -215.600,A 90.00334,B 0.00000,C 180.00000} ; release
  LIN {X 4499.921,Y 0.097,Z 84.400,A 90.00334,B 0.00000,C 180.00000} ; retreat
  ; Step 676, bar 940
  LIN {X 4515.921,Y 0.097,Z 947.280,A 90.00334,B 0.00000,C 180.00000} ; outside
  LIN {X 4515.921,Y 0.097,Z 34.400,A 90.00334,B 0.00000,C 180.00000} ; preinsert
  LIN {X 4515.921,Y 0.097,Z -215.600,A 90.00334,B 0.00000,C 180.00000} ; insert
  LIN {X 4515.921,Y 0.097,Z -215.600,A 90.00334,B 0.00000,C 180.00000} ; release
  LIN {X 4515.921,Y 0.097,Z 84.400,A 90.00334,B 0.00000,C 180.00000} ; retreat
  ; Step 677, bar 938
  LIN {X 4624.921,Y 0.097,Z 947.280,A 90.00334,B 0.00000,C 180.00000} ; outside
  LIN {X 4624.921,Y 0.097,Z 34.400,A 90.00334,B 0.00000,C 180.00000} ; preinsert
  LIN {X 4624.921,Y 0.097,Z -215.600,A 90.00334,B 0.00000,C 180.00000} ; insert
  LIN {X 4624.921,Y 0.097,Z -215.600,A 90.00334,B 0.00000,C 180.00000} ; release
  LIN {X 4624.921,Y 0.097,Z 84.400,A 90.00334,B 0.00000,C 180.00000} ; retreat
  ; Step 678, bar 941
  LIN {X 4749.921,Y 0.097,Z 947.280,A 90.00334,B 0.00000,C 180.00000} ; outside
  LIN {X 4749.921,Y 0.097,Z 34.400,A 90.00334,B 0.00000,C 180.00000} ; preinsert
  LIN {X 4749.921,Y 0.097,Z -215.600,A 90.00334,B 0.00000,C 180.00000} ; insert
  LIN {X 4749.921,Y 0.097,Z -215.600,A 90.00334,B 0.00000,C 180.00000} ; release
  LIN {X 4749.921,Y 0.097,Z 84.400,A 90.00334,B 0.00000,C 180.00000} ; retreat
  ; Step 679, bar 942
  LIN {X 4874.921,Y 0.097,Z 947.280,A 90.00334,B 0.00000,C 180.00000} ; outside
  LIN {X 4874.921,Y 0.097,Z 34.400,A 90.00334,B 0.00000,C 180.00000} ; preinsert
  LIN {X 4874.921,Y 0.097,Z -215.600,A 90.00334,B 0.00000,C 180.00000} ; insert
  LIN {X 4874.921,Y 0.097,Z -215.600,A 90.00334,B 0.00000,C 180.00000} ; release
  LIN {X 4874.921,Y 0.097,Z 84.400,A 90.00334,B 0.00000,C 180.00000} ; retreat
  ; Step 680, bar 944
  LIN {X 4999.921,Y 0.097,Z 947.280,A 90.00334,B 0.00000,C 180.00000} ; outside
  LIN {X 4999.921,Y 0.097,Z 34.400,A 90.00334,B 0.00000,C 180.00000} ; preinsert
